KUKA KRL program: EPS_2_251825_SA32_A_20260116064114.src

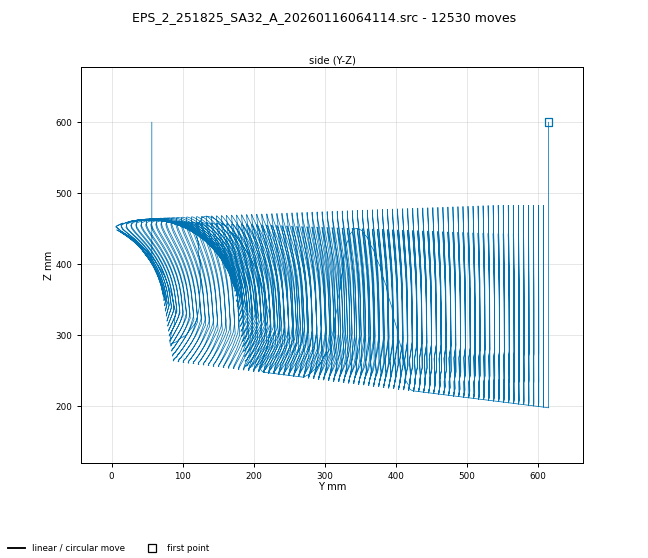
[picture p0: tool path of EPS_2_251825_SA32_A_20260116064114.src, 12530 of 12532 moves have a stored position in this frame; points joined in program order, loops and branches not executed]
&ACCESS RVP
&REL 4
&COMMENT QRS 19112012
&PARAM EDITMASK = *
DEF PART()
EXT BAS (BAS_COMMAND :IN,REAL :IN )
INT I
BAS (#INITMOV,0 )

;KUKA QRS Post kuka4.cps  Date:22-06-2017 !

File_ID=2979

QRS_PRE_INIT()

;Init var - Until changes are made in qrs_pre_init
Outlet_Square_prg=0
Inlet_1_Square_prg=0
Inlet_2_Square_prg=0
Inlet_3_Square_prg=0
Inlet_4_Square_prg=0
Inlet_5_Square_prg=0

Outlet_1={X 0.000, Y 540.910, Z 382.500, B 0.000, E1 0.000 }
Inlet_1={X 0.000, Y 543.760, Z 342.500, B 0.000, E1 213.000 }
Outlet_1_type=201
Inlet_1_type=201
;QRS#1=Sidecore dimensions
;QRS#2=200-8" PVC SDR 35
;QRS#3=200-8" PVC SDR 35
;QRS#4=
;QRS#5=
;QRS#6=
;QRS#7=
;QRS#8=
;QRS#9=12-08 PSX
;QRS#10=12-08 PSX
;QRS#11=
;QRS#12=
;QRS#13=
;QRS#14=
;QRS#15=
;QRS#16=1220x127x762 2,5'
;QRS#17=EPS Height
;QRS#18=483
;QRS#19=*
;QRS#20= UPDATED VERSION 22-06-2017
;QRS#21=*
Outlet_Square=0100
Inlet_1_Square=0100
Inlet_2_Square=0
Inlet_3_Square=0
Inlet_4_Square=0
Inlet_5_Square=0
Mill_Square=1
Outlet_Square_Prg=204
Inlet_1_Square_prg=204

QRS_INIT()

$ADVANCE=5

; T1
PTP {E1 173.659,E2 173.659}
PTP {X 0,Y 615.41,A -85,B 0,C 180,E1 173.659,E2 173.659,E3 0,E4 0,E5 0,E6 0}
QRS_SPEED_INIT()
LIN {X 0,Y 615.41,Z 600,A -85,B 0,C 180,E1 173.659,E2 173.659,E3 0,E4 0,E5 0,E6 0} C_VEL
LIN {X 0,Y 615.41,Z 207.878,A -85,B 0,C 180,E1 173.659,E2 173.659} C_VEL
LIN {X 0,Y 615.41,Z 199.7,A -85,B 0,C 180,E1 173.659,E2 173.659} C_VEL
LIN {X 0,Y 615.409,Z 197.7,A -85,B 0,C 180,E1 173.473,E2 173.473} C_VEL
LIN {X 0,Y 615.46,Z 197.7,A -85,B 0,C 180,E1 170.805,E2 170.805} C_VEL
LIN {X 0,Y 615.441,Z 197.7,A -85,B 0,C 180,E1 168.143,E2 168.143} C_VEL
LIN {X 0,Y 615.434,Z 197.7,A -85,B 0,C 180,E1 166.082,E2 166.082} C_VEL
LIN {X 0,Y 615.409,Z 197.7,A -85,B 0,C 180,E1 163.589,E2 163.589} C_VEL
LIN {X 0,Y 615.415,Z 197.7,A -85,B 0,C 180,E1 161.357,E2 161.357} C_VEL
LIN {X 0,Y 615.492,Z 197.701,A -85,B 0,C 180,E1 158.574,E2 158.574} C_VEL
LIN {X 0,Y 615.407,Z 197.7,A -85,B 0,C 180,E1 155.73,E2 155.73} C_VEL
LIN {X 0,Y 615.41,Z 197.7,A -85,B 0,C 180,E1 153.558,E2 153.558} C_VEL
LIN {X 0,Y 615.479,Z 197.703,A -85,B 0,C 180,E1 150.599,E2 150.599} C_VEL
LIN {X 0,Y 615.449,Z 197.7,A -85,B 0,C 180,E1 148.319,E2 148.319} C_VEL
LIN {X 0,Y 615.418,Z 197.7,A -85,B 0,C 180,E1 145.98,E2 145.98} C_VEL
LIN {X 0,Y 615.411,Z 197.699,A -85,B 0,C 180,E1 143.577,E2 143.577} C_VEL
LIN {X 0,Y 615.465,Z 197.699,A -85,B 0,C 180,E1 140.939,E2 140.939} C_VEL
LIN {X 0,Y 615.472,Z 197.7,A -85,B 0,C 180,E1 138.533,E2 138.533} C_VEL
LIN {X 0,Y 615.417,Z 197.7,A -85,B 0,C 180,E1 136.008,E2 136.008} C_VEL
LIN {X 0,Y 615.416,Z 197.7,A -85,B 0,C 180,E1 133.999,E2 133.999} C_VEL
LIN {X 0,Y 615.418,Z 197.699,A -85,B 0,C 180,E1 131.478,E2 131.478} C_VEL
LIN {X 0,Y 615.473,Z 197.701,A -85,B 0,C 180,E1 128.904,E2 128.904} C_VEL
LIN {X 0,Y 615.449,Z 197.7,A -85,B 0,C 180,E1 126.426,E2 126.426} C_VEL
LIN {X 0,Y 615.413,Z 197.7,A -85,B 0,C 180,E1 124.026,E2 124.026} C_VEL
LIN {X 0,Y 615.412,Z 197.699,A -85,B 0,C 180,E1 121.689,E2 121.689} C_VEL
LIN {X 0,Y 615.427,Z 197.699,A -85,B 0,C 180,E1 119.409,E2 119.409} C_VEL
LIN {X 0,Y 615.445,Z 197.7,A -85,B 0,C 180,E1 116.445,E2 116.445} C_VEL
LIN {X 0,Y 615.413,Z 197.699,A -85,B 0,C 180,E1 114.01,E2 114.01} C_VEL
LIN {X 0,Y 615.418,Z 197.7,A -85,B 0,C 180,E1 112.138,E2 112.138} C_VEL
LIN {X 0,Y 615.412,Z 197.7,A -85,B 0,C 180,E1 110.035,E2 110.035} C_VEL
LIN {X 0,Y 615.41,Z 197.7,A -85,B 0,C 180,E1 107.959,E2 107.959} C_VEL
LIN {X 0,Y 615.453,Z 197.699,A -85,B 0,C 180,E1 105.227,E2 105.227} C_VEL
LIN {X 0,Y 615.442,Z 197.701,A -85,B 0,C 180,E1 102.531,E2 102.531} C_VEL
LIN {X 0,Y 615.445,Z 197.7,A -85,B 0,C 180,E1 100.527,E2 100.527} C_VEL
LIN {X 0,Y 615.41,Z 197.7,A -85,B 0,C 180,E1 97.876,E2 97.876} C_VEL
LIN {X 0,Y 615.458,Z 197.699,A -85,B 0,C 180,E1 95.241,E2 95.241} C_VEL
LIN {X 0,Y 615.451,Z 197.7,A -85,B 0,C 180,E1 92.618,E2 92.618} C_VEL
LIN {X 0,Y 615.412,Z 197.699,A -85,B 0,C 180,E1 90,E2 90} C_VEL
LIN {X 0,Y 615.447,Z 197.699,A -85,B 0,C 180,E1 87.382,E2 87.382} C_VEL
LIN {X 0,Y 615.463,Z 197.7,A -85,B 0,C 180,E1 84.759,E2 84.759} C_VEL
LIN {X 0,Y 615.413,Z 197.699,A -85,B 0,C 180,E1 82.124,E2 82.124} C_VEL
LIN {X 0,Y 615.413,Z 197.699,A -85,B 0,C 180,E1 80.137,E2 80.137} C_VEL
LIN {X 0,Y 615.413,Z 197.699,A -85,B 0,C 180,E1 78.138,E2 78.138} C_VEL
LIN {X 0,Y 615.431,Z 197.809,A -85,B 0,C 180,E1 75.604,E2 75.604} C_VEL
LIN {X 0,Y 615.454,Z 214.764,A -85,B 0,C 180,E1 72.729,E2 72.729} C_VEL
LIN {X 0,Y 615.44,Z 229.187,A -85,B 0,C 180,E1 70.314,E2 70.314} C_VEL
LIN {X 0,Y 615.464,Z 232.183,A -85,B 0,C 180,E1 69.813,E2 69.813} C_VEL
LIN {X 0,Y 615.455,Z 338.803,A -85,B 0,C 180,E1 68.546,E2 68.546} C_VEL
LIN {X 0,Y 615.454,Z 351.86,A -85,B 0,C 180,E1 68.26,E2 68.26} C_VEL
LIN {X 0,Y 615.477,Z 364.037,A -85,B 0,C 180,E1 67.864,E2 67.864} C_VEL
LIN {X 0,Y 615.493,Z 376.068,A -85,B 0,C 180,E1 67.336,E2 67.336} C_VEL
LIN {X 0,Y 615.484,Z 387.07,A -85,B 0,C 180,E1 66.712,E2 66.712} C_VEL
LIN {X 0,Y 615.499,Z 397.482,A -85,B 0,C 180,E1 65.973,E2 65.973} C_VEL
LIN {X 0,Y 615.498,Z 406.502,A -85,B 0,C 180,E1 65.19,E2 65.19} C_VEL
LIN {X 0,Y 615.494,Z 415.026,A -85,B 0,C 180,E1 64.285,E2 64.285} C_VEL
LIN {X 0,Y 615.498,Z 422.868,A -85,B 0,C 180,E1 63.249,E2 63.249} C_VEL
LIN {X 0,Y 615.498,Z 428.792,A -85,B 0,C 180,E1 62.271,E2 62.271} C_VEL
LIN {X 0,Y 615.496,Z 433.284,A -85,B 0,C 180,E1 61.343,E2 61.343} C_VEL
LIN {X 0,Y 615.497,Z 437.518,A -85,B 0,C 180,E1 60.19,E2 60.19} C_VEL
LIN {X 0,Y 615.495,Z 440.638,A -85,B 0,C 180,E1 58.9,E2 58.9} C_VEL
LIN {X 0,Y 615.496,Z 442.14,A -85,B 0,C 180,E1 57.656,E2 57.656} C_VEL
LIN {X 0,Y 615.493,Z 442.273,A -85,B 0,C 180,E1 56.453,E2 56.453} C_VEL
LIN {X 0,Y 615.5,Z 440.932,A -85,B 0,C 180,E1 55.187,E2 55.187} C_VEL
LIN {X 0,Y 615.496,Z 438.744,A -85,B 0,C 180,E1 54.154,E2 54.154} C_VEL
LIN {X 0,Y 615.492,Z 435.237,A -85,B 0,C 180,E1 53.052,E2 53.052} C_VEL
LIN {X 0,Y 615.494,Z 430.341,A -85,B 0,C 180,E1 51.933,E2 51.933} C_VEL
LIN {X 0,Y 615.496,Z 424.633,A -85,B 0,C 180,E1 50.927,E2 50.927} C_VEL
LIN {X 0,Y 615.497,Z 417.282,A -85,B 0,C 180,E1 49.9,E2 49.9} C_VEL
LIN {X 0,Y 615.493,Z 408.29,A -85,B 0,C 180,E1 48.895,E2 48.895} C_VEL
LIN {X 0,Y 615.499,Z 399.11,A -85,B 0,C 180,E1 48.065,E2 48.065} C_VEL
LIN {X 0,Y 615.494,Z 388.597,A -85,B 0,C 180,E1 47.298,E2 47.298} C_VEL
LIN {X 0,Y 615.477,Z 377.738,A -85,B 0,C 180,E1 46.661,E2 46.661} C_VEL
LIN {X 0,Y 615.491,Z 366.43,A -85,B 0,C 180,E1 46.139,E2 46.139} C_VEL
LIN {X 0,Y 615.477,Z 353.773,A -85,B 0,C 180,E1 45.703,E2 45.703} C_VEL
LIN {X 0,Y 615.488,Z 341.141,A -85,B 0,C 180,E1 45.408,E2 45.408} C_VEL
LIN {X 0,Y 615.485,Z 319.264,A -85,B 0,C 180,E1 45.122,E2 45.122} C_VEL
LIN {X 0,Y 615.477,Z 232.126,A -85,B 0,C 180,E1 44.088,E2 44.088} C_VEL
LIN {X 0,Y 615.495,Z 215.346,A -85,B 0,C 180,E1 41.281,E2 41.281} C_VEL
LIN {X 0,Y 615.457,Z 198.823,A -85,B 0,C 180,E1 38.48,E2 38.48} C_VEL
LIN {X 0,Y 615.445,Z 197.695,A -85,B 0,C 180,E1 38.272,E2 38.272} C_VEL
LIN {X 0,Y 615.464,Z 197.689,A -85,B 0,C 180,E1 35.61,E2 35.61} C_VEL
LIN {X 0,Y 615.495,Z 197.691,A -85,B 0,C 180,E1 33.229,E2 33.229} C_VEL
LIN {X 0,Y 615.487,Z 197.702,A -85,B 0,C 180,E1 30.913,E2 30.913} C_VEL
LIN {X 0,Y 615.447,Z 197.696,A -85,B 0,C 180,E1 28.446,E2 28.446} C_VEL
LIN {X 0,Y 615.446,Z 197.696,A -85,B 0,C 180,E1 26.44,E2 26.44} C_VEL
LIN {X 0,Y 615.441,Z 197.693,A -85,B 0,C 180,E1 24.002,E2 24.002} C_VEL
LIN {X 0,Y 615.492,Z 197.689,A -85,B 0,C 180,E1 21.426,E2 21.426} C_VEL
LIN {X 0,Y 615.449,Z 197.697,A -85,B 0,C 180,E1 18.599,E2 18.599} C_VEL
LIN {X 0,Y 615.438,Z 197.696,A -85,B 0,C 180,E1 16.421,E2 16.421} C_VEL
LIN {X 0,Y 615.443,Z 197.696,A -85,B 0,C 180,E1 14.545,E2 14.545} C_VEL
LIN {X 0,Y 615.441,Z 197.696,A -85,B 0,C 180,E1 12.527,E2 12.527} C_VEL
LIN {X 0,Y 615.439,Z 197.696,A -85,B 0,C 180,E1 10.523,E2 10.523} C_VEL
LIN {X 0,Y 615.439,Z 197.696,A -85,B 0,C 180,E1 8.533,E2 8.533} C_VEL
LIN {X 0,Y 615.438,Z 197.696,A -85,B 0,C 180,E1 6.552,E2 6.552} C_VEL
LIN {X 0,Y 615.437,Z 197.697,A -85,B 0,C 180,E1 4.581,E2 4.581} C_VEL
LIN {X 0,Y 615.439,Z 197.697,A -85,B 0,C 180,E1 2.614,E2 2.614} C_VEL
LIN {X 0,Y 615.439,Z 197.697,A -85,B 0,C 180,E1 0.651,E2 0.651} C_VEL
LIN {X 0,Y 615.439,Z 197.697,A -85,B 0,C 180,E1 -1.312,E2 -1.312} C_VEL
LIN {X 0,Y 615.441,Z 197.697,A -85,B 0,C 180,E1 -3.277,E2 -3.277} C_VEL
LIN {X 0,Y 615.441,Z 197.697,A -85,B 0,C 180,E1 -5.245,E2 -5.245} C_VEL
LIN {X 0,Y 615.441,Z 197.697,A -85,B 0,C 180,E1 -7.22,E2 -7.22} C_VEL
LIN {X 0,Y 615.44,Z 197.698,A -85,B 0,C 180,E1 -9.203,E2 -9.203} C_VEL
LIN {X 0,Y 615.439,Z 197.698,A -85,B 0,C 180,E1 -11.197,E2 -11.197} C_VEL
LIN {X 0,Y 615.436,Z 197.698,A -85,B 0,C 180,E1 -13.205,E2 -13.205} C_VEL
LIN {X 0,Y 615.434,Z 197.697,A -85,B 0,C 180,E1 -15.23,E2 -15.23} C_VEL
LIN {X 0,Y 615.431,Z 197.697,A -85,B 0,C 180,E1 -17.275,E2 -17.275} C_VEL
LIN {X 0,Y 615.427,Z 197.697,A -85,B 0,C 180,E1 -19.343,E2 -19.343} C_VEL
LIN {X 0,Y 615.425,Z 197.697,A -85,B 0,C 180,E1 -21.437,E2 -21.437} C_VEL
LIN {X 0,Y 615.447,Z 197.696,A -85,B 0,C 180,E1 -24.003,E2 -24.003} C_VEL
LIN {X 0,Y 615.493,Z 197.699,A -85,B 0,C 180,E1 -26.446,E2 -26.446} C_VEL
LIN {X 0,Y 615.471,Z 197.701,A -85,B 0,C 180,E1 -28.661,E2 -28.661} C_VEL
LIN {X 0,Y 615.431,Z 197.698,A -85,B 0,C 180,E1 -31.08,E2 -31.08} C_VEL
LIN {X 0,Y 615.423,Z 197.698,A -85,B 0,C 180,E1 -33.242,E2 -33.242} C_VEL
LIN {X 0,Y 615.439,Z 197.696,A -85,B 0,C 180,E1 -35.83,E2 -35.83} C_VEL
LIN {X 0,Y 615.468,Z 197.696,A -85,B 0,C 180,E1 -38.072,E2 -38.072} C_VEL
LIN {X 0,Y 615.467,Z 197.7,A -85,B 0,C 180,E1 -40.61,E2 -40.61} C_VEL
LIN {X 0,Y 615.421,Z 197.699,A -85,B 0,C 180,E1 -43.042,E2 -43.042} C_VEL
LIN {X 0,Y 615.422,Z 197.699,A -85,B 0,C 180,E1 -45.076,E2 -45.076} C_VEL
LIN {X 0,Y 615.455,Z 197.697,A -85,B 0,C 180,E1 -47.925,E2 -47.925} C_VEL
LIN {X 0,Y 615.496,Z 197.699,A -85,B 0,C 180,E1 -50.252,E2 -50.252} C_VEL
LIN {X 0,Y 615.417,Z 197.699,A -85,B 0,C 180,E1 -53.074,E2 -53.074} C_VEL
LIN {X 0,Y 615.415,Z 197.699,A -85,B 0,C 180,E1 -55.311,E2 -55.311} C_VEL
LIN {X 0,Y 615.434,Z 197.699,A -85,B 0,C 180,E1 -57.679,E2 -57.679} C_VEL
LIN {X 0,Y 615.442,Z 197.7,A -85,B 0,C 180,E1 -60.592,E2 -60.592} C_VEL
LIN {X 0,Y 615.415,Z 197.7,A -85,B 0,C 180,E1 -62.97,E2 -62.97} C_VEL
LIN {X 0,Y 615.413,Z 197.7,A -85,B 0,C 180,E1 -65.006,E2 -65.006} C_VEL
LIN {X 0,Y 615.419,Z 197.809,A -85,B 0,C 180,E1 -67.442,E2 -67.442} C_VEL
LIN {X 0,Y 615.495,Z 217.695,A -85,B 0,C 180,E1 -70.142,E2 -70.142} C_VEL
LIN {X 0,Y 615.456,Z 238.373,A -85,B 0,C 180,E1 -72.9,E2 -72.9} C_VEL
LIN {X 0,Y 615.478,Z 258.907,A -85,B 0,C 180,E1 -75.605,E2 -75.605} C_VEL
LIN {X 0,Y 615.454,Z 270.473,A -85,B 0,C 180,E1 -77.113,E2 -77.113} C_VEL
LIN {X 0,Y 615.473,Z 378.853,A -85,B 0,C 180,E1 -78.411,E2 -78.411} C_VEL
LIN {X 0,Y 615.467,Z 391.36,A -85,B 0,C 180,E1 -78.682,E2 -78.682} C_VEL
LIN {X 0,Y 615.485,Z 404.67,A -85,B 0,C 180,E1 -79.115,E2 -79.115} C_VEL
LIN {X 0,Y 615.484,Z 416.484,A -85,B 0,C 180,E1 -79.64,E2 -79.64} C_VEL
LIN {X 0,Y 615.493,Z 427.999,A -85,B 0,C 180,E1 -80.304,E2 -80.304} C_VEL
LIN {X 0,Y 615.499,Z 438.345,A -85,B 0,C 180,E1 -81.05,E2 -81.05} C_VEL
LIN {X 0,Y 615.497,Z 446.814,A -85,B 0,C 180,E1 -81.794,E2 -81.794} C_VEL
LIN {X 0,Y 615.498,Z 454.608,A -85,B 0,C 180,E1 -82.62,E2 -82.62} C_VEL
LIN {X 0,Y 615.496,Z 462.204,A -85,B 0,C 180,E1 -83.608,E2 -83.608} C_VEL
LIN {X 0,Y 615.498,Z 469.205,A -85,B 0,C 180,E1 -84.759,E2 -84.759} C_VEL
LIN {X 0,Y 615.494,Z 473.852,A -85,B 0,C 180,E1 -85.744,E2 -85.744} C_VEL
LIN {X 0,Y 615.494,Z 477.399,A -85,B 0,C 180,E1 -86.727,E2 -86.727} C_VEL
LIN {X 0,Y 615.497,Z 479.233,A -85,B 0,C 180,E1 -87.382,E2 -87.382} C_VEL
LIN {X 0,Y 615.499,Z 480.608,A -85,B 0,C 180,E1 -88.037,E2 -88.037} C_VEL
LIN {X 0,Y 615.496,Z 482.174,A -85,B 0,C 180,E1 -89.346,E2 -89.346} C_VEL
LIN {X 0,Y 615.494,Z 482.389,A -85,B 0,C 180,E1 -90,E2 -90} C_VEL
LIN {X 0,Y 615.495,Z 481.58,A -85,B 0,C 180,E1 -91.309,E2 -91.309} C_VEL
LIN {X 0,Y 615.499,Z 480.608,A -85,B 0,C 180,E1 -91.963,E2 -91.963} C_VEL
LIN {X 0,Y 615.497,Z 479.233,A -85,B 0,C 180,E1 -92.618,E2 -92.618} C_VEL
LIN {X 0,Y 615.496,Z 476.35,A -85,B 0,C 180,E1 -93.601,E2 -93.601} C_VEL
LIN {X 0,Y 615.498,Z 472.442,A -85,B 0,C 180,E1 -94.584,E2 -94.584} C_VEL
LIN {X 0,Y 615.499,Z 467.405,A -85,B 0,C 180,E1 -95.57,E2 -95.57} C_VEL
LIN {X 0,Y 615.497,Z 460.875,A -85,B 0,C 180,E1 -96.583,E2 -96.583} C_VEL
LIN {X 0,Y 615.497,Z 453.134,A -85,B 0,C 180,E1 -97.545,E2 -97.545} C_VEL
LIN {X 0,Y 615.498,Z 445.047,A -85,B 0,C 180,E1 -98.371,E2 -98.371} C_VEL
LIN {X 0,Y 615.499,Z 435.17,A -85,B 0,C 180,E1 -99.198,E2 -99.198} C_VEL
LIN {X 0,Y 615.492,Z 423.984,A -85,B 0,C 180,E1 -99.945,E2 -99.945} C_VEL
LIN {X 0,Y 615.486,Z 413.028,A -85,B 0,C 180,E1 -100.527,E2 -100.527} C_VEL
LIN {X 0,Y 615.475,Z 400.523,A -85,B 0,C 180,E1 -101.039,E2 -101.039} C_VEL
LIN {X 0,Y 615.467,Z 388.081,A -85,B 0,C 180,E1 -101.402,E2 -101.402} C_VEL
LIN {X 0,Y 615.472,Z 374.489,A -85,B 0,C 180,E1 -101.652,E2 -101.652} C_VEL
LIN {X 0,Y 615.454,Z 270.473,A -85,B 0,C 180,E1 -102.887,E2 -102.887} C_VEL
LIN {X 0,Y 615.479,Z 249.991,A -85,B 0,C 180,E1 -105.565,E2 -105.565} C_VEL
LIN {X 0,Y 615.468,Z 228.307,A -85,B 0,C 180,E1 -108.438,E2 -108.438} C_VEL
LIN {X 0,Y 615.461,Z 209.935,A -85,B 0,C 180,E1 -110.906,E2 -110.906} C_VEL
LIN {X 0,Y 615.416,Z 197.7,A -85,B 0,C 180,E1 -112.59,E2 -112.59} C_VEL
LIN {X 0,Y 615.411,Z 197.7,A -85,B 0,C 180,E1 -114.994,E2 -114.994} C_VEL
LIN {X 0,Y 615.42,Z 197.7,A -85,B 0,C 180,E1 -117.18,E2 -117.18} C_VEL
LIN {X 0,Y 615.45,Z 197.7,A -85,B 0,C 180,E1 -120.161,E2 -120.161} C_VEL
LIN {X 0,Y 615.421,Z 197.7,A -85,B 0,C 180,E1 -122.461,E2 -122.461} C_VEL
LIN {X 0,Y 615.409,Z 197.7,A -85,B 0,C 180,E1 -124.819,E2 -124.819} C_VEL
LIN {X 0,Y 615.426,Z 197.7,A -85,B 0,C 180,E1 -127.245,E2 -127.245} C_VEL
LIN {X 0,Y 615.453,Z 197.7,A -85,B 0,C 180,E1 -130.083,E2 -130.083} C_VEL
LIN {X 0,Y 615.423,Z 197.7,A -85,B 0,C 180,E1 -132.357,E2 -132.357} C_VEL
LIN {X 0,Y 615.411,Z 197.7,A -85,B 0,C 180,E1 -134.923,E2 -134.923} C_VEL
LIN {X 0,Y 615.413,Z 197.7,A -85,B 0,C 180,E1 -136.958,E2 -136.958} C_VEL
LIN {X 0,Y 615.449,Z 197.7,A -85,B 0,C 180,E1 -139.389,E2 -139.389} C_VEL
LIN {X 0,Y 615.456,Z 197.7,A -85,B 0,C 180,E1 -141.99,E2 -141.99} C_VEL
LIN {X 0,Y 615.418,Z 197.7,A -85,B 0,C 180,E1 -144.377,E2 -144.377} C_VEL
LIN {X 0,Y 615.409,Z 197.7,A -85,B 0,C 180,E1 -146.757,E2 -146.757} C_VEL
LIN {X 0,Y 615.423,Z 197.7,A -85,B 0,C 180,E1 -149.074,E2 -149.074} C_VEL
LIN {X 0,Y 615.482,Z 197.7,A -85,B 0,C 180,E1 -151.548,E2 -151.548} C_VEL
LIN {X 0,Y 615.421,Z 197.7,A -85,B 0,C 180,E1 -154.279,E2 -154.279} C_VEL
LIN {X 0,Y 615.412,Z 197.7,A -85,B 0,C 180,E1 -156.438,E2 -156.438} C_VEL
LIN {X 0,Y 615.409,Z 197.7,A -85,B 0,C 180,E1 -158.563,E2 -158.563} C_VEL
LIN {X 0,Y 615.409,Z 197.7,A -85,B 0,C 180,E1 -160.657,E2 -160.657} C_VEL
LIN {X 0,Y 615.48,Z 197.703,A -85,B 0,C 180,E1 -163.566,E2 -163.566} C_VEL
LIN {X 0,Y 615.428,Z 197.7,A -85,B 0,C 180,E1 -166.122,E2 -166.122} C_VEL
LIN {X 0,Y 615.426,Z 197.7,A -85,B 0,C 180,E1 -168.135,E2 -168.135} C_VEL
LIN {X 0,Y 615.425,Z 197.7,A -85,B 0,C 180,E1 -170.134,E2 -170.134} C_VEL
LIN {X 0,Y 615.426,Z 197.7,A -85,B 0,C 180,E1 -172.12,E2 -172.12} C_VEL
LIN {X 0,Y 615.427,Z 197.7,A -85,B 0,C 180,E1 -174.098,E2 -174.098} C_VEL
LIN {X 0,Y 615.428,Z 197.7,A -85,B 0,C 180,E1 -176.068,E2 -176.068} C_VEL
LIN {X 0,Y 615.431,Z 197.7,A -85,B 0,C 180,E1 -178.033,E2 -178.033} C_VEL
LIN {X 0,Y 615.433,Z 197.7,A -85,B 0,C 180,E1 -179.996,E2 -179.996} C_VEL
LIN {X 0,Y 615.436,Z 197.7,A -85,B 0,C 180,E1 -181.959,E2 -181.959} C_VEL
LIN {X 0,Y 615.438,Z 197.7,A -85,B 0,C 180,E1 -183.925,E2 -183.925} C_VEL
LIN {X 0,Y 615.409,Z 197.7,A -85,B 0,C 180,E1 -186.527,E2 -186.527} C_VEL
LIN {X 0,Y 614.766,Z 197.848,A -85,B 0,C 180,E1 -187.073,E2 -187.073} C_VEL
LIN {X 0,Y 611.963,Z 198.253,A -85,B 0,C 180,E1 -187.959,E2 -187.959} C_VEL
LIN {X 0,Y 609.573,Z 198.567,A -85,B 0,C 180,E1 -188.672,E2 -188.672} C_VEL
LIN {X 0,Y 608.526,Z 198.688,A -85,B 0,C 180,E1 -189.222,E2 -189.222} C_VEL
LIN {X 0,Y 608.43,Z 198.696,A -85,B 0,C 180,E1 -189.408,E2 -189.408} C_VEL
LIN {X 0,Y 608.413,Z 198.694,A -85,B 0,C 180,E1 -191.996,E2 -191.996} C_VEL
LIN {X 0,Y 608.395,Z 198.696,A -85,B 0,C 180,E1 -194.034,E2 -194.034} C_VEL
LIN {X 0,Y 608.381,Z 198.696,A -85,B 0,C 180,E1 -196.506,E2 -196.506} C_VEL
LIN {X 0,Y 608.413,Z 198.694,A -85,B 0,C 180,E1 -198.866,E2 -198.866} C_VEL
LIN {X 0,Y 608.444,Z 198.694,A -85,B 0,C 180,E1 -201.687,E2 -201.687} C_VEL
LIN {X 0,Y 608.394,Z 198.695,A -85,B 0,C 180,E1 -204.568,E2 -204.568} C_VEL
LIN {X 0,Y 608.451,Z 198.695,A -85,B 0,C 180,E1 -207.205,E2 -207.205} C_VEL
LIN {X 0,Y 608.396,Z 198.696,A -85,B 0,C 180,E1 -209.962,E2 -209.962} C_VEL
LIN {X 0,Y 608.391,Z 198.695,A -85,B 0,C 180,E1 -212.514,E2 -212.514} C_VEL
LIN {X 0,Y 608.4,Z 198.697,A -85,B 0,C 180,E1 -214.901,E2 -214.901} C_VEL
LIN {X 0,Y 608.421,Z 198.695,A -85,B 0,C 180,E1 -217.742,E2 -217.742} C_VEL
LIN {X 0,Y 608.382,Z 198.696,A -85,B 0,C 180,E1 -220.323,E2 -220.323} C_VEL
LIN {X 0,Y 608.424,Z 198.696,A -85,B 0,C 180,E1 -222.954,E2 -222.954} C_VEL
LIN {X 0,Y 608.4,Z 198.697,A -85,B 0,C 180,E1 -225.733,E2 -225.733} C_VEL
LIN {X 0,Y 608.401,Z 198.695,A -85,B 0,C 180,E1 -227.935,E2 -227.935} C_VEL
LIN {X 0,Y 608.428,Z 198.693,A -85,B 0,C 180,E1 -230.697,E2 -230.697} C_VEL
LIN {X 0,Y 608.434,Z 198.698,A -85,B 0,C 180,E1 -233.085,E2 -233.085} C_VEL
LIN {X 0,Y 608.441,Z 198.694,A -85,B 0,C 180,E1 -235.53,E2 -235.53} C_VEL
LIN {X 0,Y 608.409,Z 198.694,A -85,B 0,C 180,E1 -237.903,E2 -237.903} C_VEL
LIN {X 0,Y 608.396,Z 198.694,A -85,B 0,C 180,E1 -240.217,E2 -240.217} C_VEL
LIN {X 0,Y 608.44,Z 198.693,A -85,B 0,C 180,E1 -242.785,E2 -242.785} C_VEL
LIN {X 0,Y 608.411,Z 198.693,A -85,B 0,C 180,E1 -245.845,E2 -245.845} C_VEL
LIN {X 0,Y 608.406,Z 198.693,A -85,B 0,C 180,E1 -248.307,E2 -248.307} C_VEL
LIN {X 0,Y 608.431,Z 198.701,A -85,B 0,C 180,E1 -251.13,E2 -251.13} C_VEL
LIN {X 0,Y 608.396,Z 198.695,A -85,B 0,C 180,E1 -253.905,E2 -253.905} C_VEL
LIN {X 0,Y 608.42,Z 198.694,A -85,B 0,C 180,E1 -256.643,E2 -256.643} C_VEL
LIN {X 0,Y 608.431,Z 198.696,A -85,B 0,C 180,E1 -259.35,E2 -259.35} C_VEL
LIN {X 0,Y 608.406,Z 198.693,A -85,B 0,C 180,E1 -262.032,E2 -262.032} C_VEL
LIN {X 0,Y 608.431,Z 198.694,A -85,B 0,C 180,E1 -264.698,E2 -264.698} C_VEL
LIN {X 0,Y 608.439,Z 198.694,A -85,B 0,C 180,E1 -267.352,E2 -267.352} C_VEL
LIN {X 0,Y 608.403,Z 198.693,A -85,B 0,C 180,E1 -270,E2 -270} C_VEL
LIN {X 0,Y 608.436,Z 198.694,A -85,B 0,C 180,E1 -272.648,E2 -272.648} C_VEL
LIN {X 0,Y 608.435,Z 198.695,A -85,B 0,C 180,E1 -275.302,E2 -275.302} C_VEL
LIN {X 0,Y 608.408,Z 198.693,A -85,B 0,C 180,E1 -277.968,E2 -277.968} C_VEL
LIN {X 0,Y 608.429,Z 198.695,A -85,B 0,C 180,E1 -280.65,E2 -280.65} C_VEL
LIN {X 0,Y 608.426,Z 198.695,A -85,B 0,C 180,E1 -283.357,E2 -283.357} C_VEL
LIN {X 0,Y 608.438,Z 198.817,A -85,B 0,C 180,E1 -284.336,E2 -284.336} C_VEL
LIN {X 0,Y 608.443,Z 216.169,A -85,B 0,C 180,E1 -287.303,E2 -287.303} C_VEL
LIN {X 0,Y 608.419,Z 230.661,A -85,B 0,C 180,E1 -289.747,E2 -289.747} C_VEL
LIN {X 0,Y 608.43,Z 232.362,A -85,B 0,C 180,E1 -290.032,E2 -290.032} C_VEL
LIN {X 0,Y 608.536,Z 331.818,A -85,B 0,C 180,E1 -291.222,E2 -291.222} C_VEL
LIN {X 0,Y 608.503,Z 345.333,A -85,B 0,C 180,E1 -291.445,E2 -291.445} C_VEL
LIN {X 0,Y 608.492,Z 359.013,A -85,B 0,C 180,E1 -291.824,E2 -291.824} C_VEL
LIN {X 0,Y 608.506,Z 371.463,A -85,B 0,C 180,E1 -292.314,E2 -292.314} C_VEL
LIN {X 0,Y 608.483,Z 383.511,A -85,B 0,C 180,E1 -292.945,E2 -292.945} C_VEL
LIN {X 0,Y 608.497,Z 394.341,A -85,B 0,C 180,E1 -293.662,E2 -293.662} C_VEL
LIN {X 0,Y 608.478,Z 403.986,A -85,B 0,C 180,E1 -294.45,E2 -294.45} C_VEL
LIN {X 0,Y 608.451,Z 412.483,A -85,B 0,C 180,E1 -295.3,E2 -295.3} C_VEL
LIN {X 0,Y 608.46,Z 420.032,A -85,B 0,C 180,E1 -296.218,E2 -296.218} C_VEL
LIN {X 0,Y 608.453,Z 426.713,A -85,B 0,C 180,E1 -297.217,E2 -297.217} C_VEL
LIN {X 0,Y 608.441,Z 432.294,A -85,B 0,C 180,E1 -298.266,E2 -298.266} C_VEL
LIN {X 0,Y 608.426,Z 436.889,A -85,B 0,C 180,E1 -299.4,E2 -299.4} C_VEL
LIN {X 0,Y 608.446,Z 440.145,A -85,B 0,C 180,E1 -300.545,E2 -300.545} C_VEL
LIN {X 0,Y 608.441,Z 441.63,A -85,B 0,C 180,E1 -301.317,E2 -301.317} C_VEL
LIN {X 0,Y 608.421,Z 442.879,A -85,B 0,C 180,E1 -302.529,E2 -302.529} C_VEL
LIN {X 0,Y 608.416,Z 442.761,A -85,B 0,C 180,E1 -303.739,E2 -303.739} C_VEL
LIN {X 0,Y 608.424,Z 441.396,A -85,B 0,C 180,E1 -304.913,E2 -304.913} C_VEL
LIN {X 0,Y 608.443,Z 438.748,A -85,B 0,C 180,E1 -306.091,E2 -306.091} C_VEL
LIN {X 0,Y 608.43,Z 435.136,A -85,B 0,C 180,E1 -307.164,E2 -307.164} C_VEL
LIN {X 0,Y 608.431,Z 430.227,A -85,B 0,C 180,E1 -308.246,E2 -308.246} C_VEL
LIN {X 0,Y 608.441,Z 424.013,A -85,B 0,C 180,E1 -309.304,E2 -309.304} C_VEL
LIN {X 0,Y 608.457,Z 416.373,A -85,B 0,C 180,E1 -310.339,E2 -310.339} C_VEL
LIN {X 0,Y 608.452,Z 408.826,A -85,B 0,C 180,E1 -311.175,E2 -311.175} C_VEL
LIN {X 0,Y 608.495,Z 399.125,A -85,B 0,C 180,E1 -312.057,E2 -312.057} C_VEL
LIN {X 0,Y 608.505,Z 387.951,A -85,B 0,C 180,E1 -312.87,E2 -312.87} C_VEL
LIN {X 0,Y 608.498,Z 376.576,A -85,B 0,C 180,E1 -313.529,E2 -313.529} C_VEL
LIN {X 0,Y 608.507,Z 364.752,A -85,B 0,C 180,E1 -314.058,E2 -314.058} C_VEL
LIN {X 0,Y 608.539,Z 351.382,A -85,B 0,C 180,E1 -314.496,E2 -314.496} C_VEL
LIN {X 0,Y 608.547,Z 338.609,A -85,B 0,C 180,E1 -314.774,E2 -314.774} C_VEL
LIN {X 0,Y 608.463,Z 232.347,A -85,B 0,C 180,E1 -316.059,E2 -316.059} C_VEL
LIN {X 0,Y 608.475,Z 215.893,A -85,B 0,C 180,E1 -318.833,E2 -318.833} C_VEL
LIN {X 0,Y 608.479,Z 200.746,A -85,B 0,C 180,E1 -321.42,E2 -321.42} C_VEL
LIN {X 0,Y 608.416,Z 198.694,A -85,B 0,C 180,E1 -321.794,E2 -321.794} C_VEL
LIN {X 0,Y 608.435,Z 198.69,A -85,B 0,C 180,E1 -323.954,E2 -323.954} C_VEL
LIN {X 0,Y 608.439,Z 198.69,A -85,B 0,C 180,E1 -326.335,E2 -326.335} C_VEL
LIN {X 0,Y 608.451,Z 198.693,A -85,B 0,C 180,E1 -328.729,E2 -328.729} C_VEL
LIN {X 0,Y 608.442,Z 198.693,A -85,B 0,C 180,E1 -331.383,E2 -331.383} C_VEL
LIN {X 0,Y 608.436,Z 198.696,A -85,B 0,C 180,E1 -333.231,E2 -333.231} C_VEL
LIN {X 0,Y 608.435,Z 198.69,A -85,B 0,C 180,E1 -335.853,E2 -335.853} C_VEL
LIN {X 0,Y 608.452,Z 198.689,A -85,B 0,C 180,E1 -338.313,E2 -338.313} C_VEL
LIN {X 0,Y 608.438,Z 198.694,A -85,B 0,C 180,E1 -341.289,E2 -341.289} C_VEL
LIN {X 0,Y 608.418,Z 198.692,A -85,B 0,C 180,E1 -343.91,E2 -343.91} C_VEL
LIN {X 0,Y 608.46,Z 198.693,A -85,B 0,C 180,E1 -346.648,E2 -346.648} C_VEL
LIN {X 0,Y 608.428,Z 198.693,A -85,B 0,C 180,E1 -349.354,E2 -349.354} C_VEL
LIN {X 0,Y 608.443,Z 198.689,A -85,B 0,C 180,E1 -352.037,E2 -352.037} C_VEL
LIN {X 0,Y 608.467,Z 198.694,A -85,B 0,C 180,E1 -354.702,E2 -354.702} C_VEL
LIN {X 0,Y 608.435,Z 198.691,A -85,B 0,C 180,E1 -357.356,E2 -357.356} C_VEL
LIN {X 0,Y 608.437,Z 198.691,A -85,B 0,C 180,E1 -359.342,E2 -359.342} C_VEL
LIN {X 0,Y 608.426,Z 198.692,A -85,B 0,C 180,E1 -361.327,E2 -361.327} C_VEL
LIN {X 0,Y 608.409,Z 198.695,A -85,B 0,C 180,E1 -363.315,E2 -363.315} C_VEL
LIN {X 0,Y 608.422,Z 198.693,A -85,B 0,C 180,E1 -365.306,E2 -365.306} C_VEL
LIN {X 0,Y 608.412,Z 198.694,A -85,B 0,C 180,E1 -367.303,E2 -367.303} C_VEL
LIN {X 0,Y 608.426,Z 198.692,A -85,B 0,C 180,E1 -369.31,E2 -369.31} C_VEL
LIN {X 0,Y 608.411,Z 198.694,A -85,B 0,C 180,E1 -371.328,E2 -371.328} C_VEL
LIN {X 0,Y 608.417,Z 198.692,A -85,B 0,C 180,E1 -373.361,E2 -373.361} C_VEL
LIN {X 0,Y 608.425,Z 198.691,A -85,B 0,C 180,E1 -375.41,E2 -375.41} C_VEL
LIN {X 0,Y 608.407,Z 198.693,A -85,B 0,C 180,E1 -377.481,E2 -377.481} C_VEL
LIN {X 0,Y 608.407,Z 198.693,A -85,B 0,C 180,E1 -379.575,E2 -379.575} C_VEL
LIN {X 0,Y 608.425,Z 198.691,A -85,B 0,C 180,E1 -381.696,E2 -381.696} C_VEL
LIN {X 0,Y 608.434,Z 198.7,A -85,B 0,C 180,E1 -384.574,E2 -384.574} C_VEL
LIN {X 0,Y 608.413,Z 198.693,A -85,B 0,C 180,E1 -387.198,E2 -387.198} C_VEL
LIN {X 0,Y 608.405,Z 198.696,A -85,B 0,C 180,E1 -389.026,E2 -389.026} C_VEL
LIN {X 0,Y 608.404,Z 198.693,A -85,B 0,C 180,E1 -391.322,E2 -391.322} C_VEL
LIN {X 0,Y 608.423,Z 198.692,A -85,B 0,C 180,E1 -393.73,E2 -393.73} C_VEL
LIN {X 0,Y 608.436,Z 198.694,A -85,B 0,C 180,E1 -396.095,E2 -396.095} C_VEL
LIN {X 0,Y 608.405,Z 198.701,A -85,B 0,C 180,E1 -398.595,E2 -398.595} C_VEL
LIN {X 0,Y 608.392,Z 198.695,A -85,B 0,C 180,E1 -401.184,E2 -401.184} C_VEL
LIN {X 0,Y 608.413,Z 198.692,A -85,B 0,C 180,E1 -403.305,E2 -403.305} C_VEL
LIN {X 0,Y 608.449,Z 198.695,A -85,B 0,C 180,E1 -406.13,E2 -406.13} C_VEL
LIN {X 0,Y 608.406,Z 198.696,A -85,B 0,C 180,E1 -408.821,E2 -408.821} C_VEL
LIN {X 0,Y 608.39,Z 198.695,A -85,B 0,C 180,E1 -411.407,E2 -411.407} C_VEL
LIN {X 0,Y 608.44,Z 198.694,A -85,B 0,C 180,E1 -413.957,E2 -413.957} C_VEL
LIN {X 0,Y 608.445,Z 198.698,A -85,B 0,C 180,E1 -416.329,E2 -416.329} C_VEL
LIN {X 0,Y 608.426,Z 198.693,A -85,B 0,C 180,E1 -418.737,E2 -418.737} C_VEL
LIN {X 0,Y 608.388,Z 198.696,A -85,B 0,C 180,E1 -420.977,E2 -420.977} C_VEL
LIN {X 0,Y 608.383,Z 198.696,A -85,B 0,C 180,E1 -423.223,E2 -423.223} C_VEL
LIN {X 0,Y 608.406,Z 198.694,A -85,B 0,C 180,E1 -425.428,E2 -425.428} C_VEL
LIN {X 0,Y 608.415,Z 198.825,A -85,B 0,C 180,E1 -427.309,E2 -427.309} C_VEL
LIN {X 0,Y 608.538,Z 212.666,A -85,B 0,C 180,E1 -429.218,E2 -429.218} C_VEL
LIN {X 0,Y 608.509,Z 231.945,A -85,B 0,C 180,E1 -431.831,E2 -431.831} C_VEL
LIN {X 0,Y 608.477,Z 252.656,A -85,B 0,C 180,E1 -434.595,E2 -434.595} C_VEL
LIN {X 0,Y 608.441,Z 270.616,A -85,B 0,C 180,E1 -436.962,E2 -436.962} C_VEL
LIN {X 0,Y 608.571,Z 337.355,A -85,B 0,C 180,E1 -437.77,E2 -437.77} C_VEL
LIN {X 0,Y 608.526,Z 380.108,A -85,B 0,C 180,E1 -438.298,E2 -438.298} C_VEL
LIN {X 0,Y 608.517,Z 393.748,A -85,B 0,C 180,E1 -438.614,E2 -438.614} C_VEL
LIN {X 0,Y 608.509,Z 405.819,A -85,B 0,C 180,E1 -439.027,E2 -439.027} C_VEL
LIN {X 0,Y 608.494,Z 418.212,A -85,B 0,C 180,E1 -439.603,E2 -439.603} C_VEL
LIN {X 0,Y 608.506,Z 429.479,A -85,B 0,C 180,E1 -440.276,E2 -440.276} C_VEL
LIN {X 0,Y 608.474,Z 439.65,A -85,B 0,C 180,E1 -441.03,E2 -441.03} C_VEL
LIN {X 0,Y 608.464,Z 448.79,A -85,B 0,C 180,E1 -441.866,E2 -441.866} C_VEL
LIN {X 0,Y 608.466,Z 457.692,A -85,B 0,C 180,E1 -442.868,E2 -442.868} C_VEL
LIN {X 0,Y 608.443,Z 464.851,A -85,B 0,C 180,E1 -443.867,E2 -443.867} C_VEL
LIN {X 0,Y 608.463,Z 469.681,A -85,B 0,C 180,E1 -444.698,E2 -444.698} C_VEL
LIN {X 0,Y 608.439,Z 474.371,A -85,B 0,C 180,E1 -445.694,E2 -445.694} C_VEL
LIN {X 0,Y 608.424,Z 477.956,A -85,B 0,C 180,E1 -446.689,E2 -446.689} C_VEL
LIN {X 0,Y 608.425,Z 479.809,A -85,B 0,C 180,E1 -447.352,E2 -447.352} C_VEL
LIN {X 0,Y 608.444,Z 481.201,A -85,B 0,C 180,E1 -448.014,E2 -448.014} C_VEL
LIN {X 0,Y 608.439,Z 482.783,A -85,B 0,C 180,E1 -449.338,E2 -449.338} C_VEL
LIN {X 0,Y 608.434,Z 483,A -85,B 0,C 180,E1 -450,E2 -450} C_VEL
LIN {X 0,Y 608.448,Z 482.184,A -85,B 0,C 180,E1 -451.324,E2 -451.324} C_VEL
LIN {X 0,Y 608.444,Z 481.201,A -85,B 0,C 180,E1 -451.986,E2 -451.986} C_VEL
LIN {X 0,Y 608.425,Z 479.809,A -85,B 0,C 180,E1 -452.648,E2 -452.648} C_VEL
LIN {X 0,Y 608.449,Z 476.896,A -85,B 0,C 180,E1 -453.642,E2 -453.642} C_VEL
LIN {X 0,Y 608.432,Z 472.95,A -85,B 0,C 180,E1 -454.638,E2 -454.638} C_VEL
LIN {X 0,Y 608.437,Z 466.877,A -85,B 0,C 180,E1 -455.801,E2 -455.801} C_VEL
LIN {X 0,Y 608.463,Z 460.236,A -85,B 0,C 180,E1 -456.799,E2 -456.799} C_VEL
LIN {X 0,Y 608.456,Z 451.991,A -85,B 0,C 180,E1 -457.8,E2 -457.8} C_VEL
LIN {X 0,Y 608.472,Z 443.538,A -85,B 0,C 180,E1 -458.636,E2 -458.636} C_VEL
LIN {X 0,Y 608.479,Z 433.094,A -85,B 0,C 180,E1 -459.473,E2 -459.473} C_VEL
LIN {X 0,Y 608.498,Z 422.76,A -85,B 0,C 180,E1 -460.144,E2 -460.144} C_VEL
LIN {X 0,Y 608.517,Z 411.61,A -85,B 0,C 180,E1 -460.724,E2 -460.724} C_VEL
LIN {X 0,Y 608.517,Z 399.912,A -85,B 0,C 180,E1 -461.192,E2 -461.192} C_VEL
LIN {X 0,Y 608.53,Z 387.278,A -85,B 0,C 180,E1 -461.555,E2 -461.555} C_VEL
LIN {X 0,Y 608.534,Z 374.62,A -85,B 0,C 180,E1 -461.787,E2 -461.787} C_VEL
LIN {X 0,Y 608.496,Z 271.168,A -85,B 0,C 180,E1 -463.016,E2 -463.016} C_VEL
LIN {X 0,Y 608.444,Z 270.13,A -85,B 0,C 180,E1 -463.102,E2 -463.102} C_VEL
LIN {X 0,Y 608.495,Z 250.066,A -85,B 0,C 180,E1 -465.748,E2 -465.748} C_VEL
LIN {X 0,Y 608.514,Z 229.536,A -85,B 0,C 180,E1 -468.494,E2 -468.494} C_VEL
LIN {X 0,Y 608.54,Z 209.939,A -85,B 0,C 180,E1 -471.155,E2 -471.155} C_VEL
LIN {X 0,Y 608.404,Z 198.695,A -85,B 0,C 180,E1 -472.716,E2 -472.716} C_VEL
LIN {X 0,Y 608.399,Z 198.696,A -85,B 0,C 180,E1 -475.303,E2 -475.303} C_VEL
LIN {X 0,Y 608.404,Z 198.697,A -85,B 0,C 180,E1 -478.268,E2 -478.268} C_VEL
LIN {X 0,Y 608.401,Z 198.694,A -85,B 0,C 180,E1 -480.548,E2 -480.548} C_VEL
LIN {X 0,Y 608.406,Z 198.693,A -85,B 0,C 180,E1 -482.882,E2 -482.882} C_VEL
LIN {X 0,Y 608.409,Z 198.695,A -85,B 0,C 180,E1 -485.279,E2 -485.279} C_VEL
LIN {X 0,Y 608.408,Z 198.696,A -85,B 0,C 180,E1 -488.231,E2 -488.231} C_VEL
LIN {X 0,Y 608.404,Z 198.695,A -85,B 0,C 180,E1 -490.322,E2 -490.322} C_VEL
LIN {X 0,Y 608.383,Z 198.696,A -85,B 0,C 180,E1 -492.965,E2 -492.965} C_VEL
LIN {X 0,Y 608.446,Z 198.699,A -85,B 0,C 180,E1 -495.736,E2 -495.736} C_VEL
LIN {X 0,Y 608.451,Z 198.694,A -85,B 0,C 180,E1 -497.936,E2 -497.936} C_VEL
LIN {X 0,Y 608.396,Z 198.694,A -85,B 0,C 180,E1 -500.553,E2 -500.553} C_VEL
LIN {X 0,Y 608.389,Z 198.697,A -85,B 0,C 180,E1 -503.078,E2 -503.078} C_VEL
LIN {X 0,Y 608.434,Z 198.697,A -85,B 0,C 180,E1 -505.526,E2 -505.526} C_VEL
LIN {X 0,Y 608.448,Z 198.695,A -85,B 0,C 180,E1 -507.902,E2 -507.902} C_VEL
LIN {X 0,Y 608.416,Z 198.694,A -85,B 0,C 180,E1 -510.215,E2 -510.215} C_VEL
LIN {X 0,Y 608.398,Z 198.694,A -85,B 0,C 180,E1 -512.805,E2 -512.805} C_VEL
LIN {X 0,Y 608.425,Z 198.698,A -85,B 0,C 180,E1 -515.425,E2 -515.425} C_VEL
LIN {X 0,Y 608.416,Z 198.693,A -85,B 0,C 180,E1 -518.304,E2 -518.304} C_VEL
LIN {X 0,Y 608.394,Z 198.695,A -85,B 0,C 180,E1 -520.425,E2 -520.425} C_VEL
LIN {X 0,Y 608.417,Z 198.696,A -85,B 0,C 180,E1 -523.212,E2 -523.212} C_VEL
LIN {X 0,Y 608.421,Z 198.695,A -85,B 0,C 180,E1 -525.996,E2 -525.996} C_VEL
LIN {X 0,Y 608.417,Z 198.695,A -85,B 0,C 180,E1 -527.996,E2 -527.996} C_VEL
LIN {X 0,Y 608.409,Z 198.696,A -85,B 0,C 180,E1 -530.019,E2 -530.019} C_VEL
LIN {X 0,Y 608.394,Z 198.695,A -85,B 0,C 180,E1 -532.696,E2 -532.696} C_VEL
LIN {X 0,Y 608.443,Z 198.696,A -85,B 0,C 180,E1 -535.359,E2 -535.359} C_VEL
LIN {X 0,Y 608.404,Z 198.696,A -85,B 0,C 180,E1 -538.01,E2 -538.01} C_VEL
LIN {X 0,Y 608.427,Z 198.693,A -85,B 0,C 180,E1 -539.996,E2 -539.996} C_VEL
LIN {X 0,Y 608.409,Z 198.693,A -85,B 0,C 180,E1 -542.644,E2 -542.644} C_VEL
LIN {X 0,Y 608.44,Z 198.696,A -85,B 0,C 180,E1 -545.298,E2 -545.298} C_VEL
LIN {X 0,Y 608.401,Z 198.696,A -85,B 0,C 180,E1 -547.964,E2 -547.964} C_VEL
LIN {X 0,Y 608.43,Z 198.696,A -85,B 0,C 180,E1 -549.408,E2 -549.408} C_VEL
LIN {X 0,Y 607.738,Z 198.779,A -85,B 0,C 180,E1 -549.96,E2 -549.96} C_VEL
LIN {X 0,Y 604.883,Z 199.134,A -85,B 0,C 180,E1 -550.857,E2 -550.857} C_VEL
LIN {X 0,Y 602.481,Z 199.44,A -85,B 0,C 180,E1 -551.579,E2 -551.579} C_VEL
LIN {X 0,Y 601.442,Z 199.562,A -85,B 0,C 180,E1 -552.135,E2 -552.135} C_VEL
LIN {X 0,Y 601.352,Z 199.572,A -85,B 0,C 180,E1 -552.324,E2 -552.324} C_VEL
LIN {X 0,Y 601.365,Z 199.572,A -85,B 0,C 180,E1 -554.894,E2 -554.894} C_VEL
LIN {X 0,Y 601.361,Z 199.577,A -85,B 0,C 180,E1 -557.684,E2 -557.684} C_VEL
LIN {X 0,Y 601.364,Z 199.574,A -85,B 0,C 180,E1 -559.806,E2 -559.806} C_VEL
LIN {X 0,Y 601.368,Z 199.57,A -85,B 0,C 180,E1 -562.679,E2 -562.679} C_VEL
LIN {X 0,Y 601.401,Z 199.572,A -85,B 0,C 180,E1 -565.613,E2 -565.613} C_VEL
LIN {X 0,Y 601.353,Z 199.574,A -85,B 0,C 180,E1 -567.865,E2 -567.865} C_VEL
LIN {X 0,Y 601.36,Z 199.571,A -85,B 0,C 180,E1 -570.161,E2 -570.161} C_VEL
LIN {X 0,Y 601.367,Z 199.571,A -85,B 0,C 180,E1 -572.709,E2 -572.709} C_VEL
LIN {X 0,Y 601.354,Z 199.578,A -85,B 0,C 180,E1 -575.108,E2 -575.108} C_VEL
LIN {X 0,Y 601.394,Z 199.576,A -85,B 0,C 180,E1 -577.415,E2 -577.415} C_VEL
LIN {X 0,Y 601.364,Z 199.571,A -85,B 0,C 180,E1 -579.991,E2 -579.991} C_VEL
LIN {X 0,Y 601.362,Z 199.572,A -85,B 0,C 180,E1 -582.666,E2 -582.666} C_VEL
LIN {X 0,Y 601.373,Z 199.576,A -85,B 0,C 180,E1 -585.478,E2 -585.478} C_VEL
LIN {X 0,Y 601.366,Z 199.57,A -85,B 0,C 180,E1 -588.231,E2 -588.231} C_VEL
LIN {X 0,Y 601.389,Z 199.571,A -85,B 0,C 180,E1 -590.873,E2 -590.873} C_VEL
LIN {X 0,Y 601.39,Z 199.57,A -85,B 0,C 180,E1 -593.73,E2 -593.73} C_VEL
LIN {X 0,Y 601.36,Z 199.571,A -85,B 0,C 180,E1 -596.063,E2 -596.063} C_VEL
LIN {X 0,Y 601.384,Z 199.569,A -85,B 0,C 180,E1 -598.538,E2 -598.538} C_VEL
LIN {X 0,Y 601.402,Z 199.573,A -85,B 0,C 180,E1 -601.372,E2 -601.372} C_VEL
LIN {X 0,Y 601.355,Z 199.575,A -85,B 0,C 180,E1 -603.635,E2 -603.635} C_VEL
LIN {X 0,Y 601.368,Z 199.572,A -85,B 0,C 180,E1 -606.588,E2 -606.588} C_VEL
LIN {X 0,Y 601.394,Z 199.571,A -85,B 0,C 180,E1 -609.477,E2 -609.477} C_VEL
LIN {X 0,Y 601.342,Z 199.573,A -85,B 0,C 180,E1 -612.31,E2 -612.31} C_VEL
LIN {X 0,Y 601.363,Z 199.571,A -85,B 0,C 180,E1 -614.408,E2 -614.408} C_VEL
LIN {X 0,Y 601.377,Z 199.578,A -85,B 0,C 180,E1 -617.171,E2 -617.171} C_VEL
LIN {X 0,Y 601.394,Z 199.575,A -85,B 0,C 180,E1 -619.224,E2 -619.224} C_VEL
LIN {X 0,Y 601.373,Z 199.569,A -85,B 0,C 180,E1 -621.938,E2 -621.938} C_VEL
LIN {X 0,Y 601.346,Z 199.572,A -85,B 0,C 180,E1 -623.962,E2 -623.962} C_VEL
LIN {X 0,Y 601.392,Z 199.571,A -85,B 0,C 180,E1 -626.65,E2 -626.65} C_VEL
LIN {X 0,Y 601.412,Z 199.57,A -85,B 0,C 180,E1 -629.33,E2 -629.33} C_VEL
LIN {X 0,Y 601.354,Z 199.571,A -85,B 0,C 180,E1 -632.009,E2 -632.009} C_VEL
LIN {X 0,Y 601.38,Z 199.573,A -85,B 0,C 180,E1 -634.692,E2 -634.692} C_VEL
LIN {X 0,Y 601.402,Z 199.57,A -85,B 0,C 180,E1 -637.385,E2 -637.385} C_VEL
LIN {X 0,Y 601.371,Z 199.57,A -85,B 0,C 180,E1 -640.096,E2 -640.096} C_VEL
LIN {X 0,Y 601.356,Z 199.572,A -85,B 0,C 180,E1 -642.143,E2 -642.143} C_VEL
LIN {X 0,Y 601.371,Z 199.626,A -85,B 0,C 180,E1 -644.249,E2 -644.249} C_VEL
LIN {X 0,Y 601.433,Z 213.458,A -85,B 0,C 180,E1 -646.648,E2 -646.648} C_VEL
LIN {X 0,Y 601.4,Z 228.822,A -85,B 0,C 180,E1 -649.276,E2 -649.276} C_VEL
LIN {X 0,Y 601.363,Z 232.364,A -85,B 0,C 180,E1 -649.877,E2 -649.877} C_VEL
LIN {X 0,Y 601.656,Z 237.586,A -85,B 0,C 180,E1 -649.956,E2 -649.956} C_VEL
LIN {X 0,Y 601.579,Z 339.131,A -85,B 0,C 180,E1 -651.187,E2 -651.187} C_VEL
LIN {X 0,Y 601.555,Z 352.135,A -85,B 0,C 180,E1 -651.48,E2 -651.48} C_VEL
LIN {X 0,Y 601.545,Z 364.903,A -85,B 0,C 180,E1 -651.908,E2 -651.908} C_VEL
LIN {X 0,Y 601.511,Z 375.966,A -85,B 0,C 180,E1 -652.407,E2 -652.407} C_VEL
LIN {X 0,Y 601.449,Z 387.052,A -85,B 0,C 180,E1 -653.044,E2 -653.044} C_VEL
LIN {X 0,Y 601.466,Z 398.348,A -85,B 0,C 180,E1 -653.864,E2 -653.864} C_VEL
LIN {X 0,Y 601.428,Z 407.834,A -85,B 0,C 180,E1 -654.716,E2 -654.716} C_VEL
LIN {X 0,Y 601.384,Z 417.048,A -85,B 0,C 180,E1 -655.748,E2 -655.748} C_VEL
LIN {X 0,Y 601.357,Z 424.197,A -85,B 0,C 180,E1 -656.739,E2 -656.739} C_VEL
LIN {X 0,Y 601.343,Z 430.664,A -85,B 0,C 180,E1 -657.87,E2 -657.87} C_VEL
LIN {X 0,Y 601.328,Z 435.824,A -85,B 0,C 180,E1 -659.064,E2 -659.064} C_VEL
LIN {X 0,Y 601.355,Z 439.288,A -85,B 0,C 180,E1 -660.167,E2 -660.167} C_VEL
LIN {X 0,Y 601.353,Z 441.887,A -85,B 0,C 180,E1 -661.457,E2 -661.457} C_VEL
LIN {X 0,Y 601.322,Z 442.929,A -85,B 0,C 180,E1 -662.713,E2 -662.713} C_VEL
LIN {X 0,Y 601.31,Z 442.634,A -85,B 0,C 180,E1 -663.93,E2 -663.93} C_VEL
LIN {X 0,Y 601.319,Z 441.104,A -85,B 0,C 180,E1 -665.113,E2 -665.113} C_VEL
LIN {X 0,Y 601.342,Z 438.369,A -85,B 0,C 180,E1 -666.264,E2 -666.264} C_VEL
LIN {X 0,Y 601.367,Z 434.281,A -85,B 0,C 180,E1 -667.423,E2 -667.423} C_VEL
LIN {X 0,Y 601.337,Z 429.357,A -85,B 0,C 180,E1 -668.47,E2 -668.47} C_VEL
LIN {X 0,Y 601.378,Z 422.945,A -85,B 0,C 180,E1 -669.539,E2 -669.539} C_VEL
LIN {X 0,Y 601.412,Z 415.1,A -85,B 0,C 180,E1 -670.583,E2 -670.583} C_VEL
LIN {X 0,Y 601.418,Z 406.957,A -85,B 0,C 180,E1 -671.459,E2 -671.459} C_VEL
LIN {X 0,Y 601.454,Z 397.296,A -85,B 0,C 180,E1 -672.31,E2 -672.31} C_VEL
LIN {X 0,Y 601.495,Z 387.676,A -85,B 0,C 180,E1 -673.004,E2 -673.004} C_VEL
LIN {X 0,Y 601.511,Z 376.218,A -85,B 0,C 180,E1 -673.671,E2 -673.671} C_VEL
LIN {X 0,Y 601.522,Z 364.811,A -85,B 0,C 180,E1 -674.186,E2 -674.186} C_VEL
LIN {X 0,Y 601.557,Z 352.14,A -85,B 0,C 180,E1 -674.61,E2 -674.61} C_VEL
LIN {X 0,Y 601.604,Z 338.691,A -85,B 0,C 180,E1 -674.91,E2 -674.91} C_VEL
LIN {X 0,Y 601.634,Z 233.749,A -85,B 0,C 180,E1 -676.181,E2 -676.181} C_VEL
LIN {X 0,Y 601.426,Z 232.317,A -85,B 0,C 180,E1 -676.22,E2 -676.22} C_VEL
LIN {X 0,Y 601.451,Z 216.283,A -85,B 0,C 180,E1 -678.955,E2 -678.955} C_VEL
LIN {X 0,Y 601.476,Z 201.435,A -85,B 0,C 180,E1 -681.522,E2 -681.522} C_VEL
LIN {X 0,Y 601.413,Z 199.567,A -85,B 0,C 180,E1 -681.872,E2 -681.872} C_VEL
LIN {X 0,Y 601.414,Z 199.571,A -85,B 0,C 180,E1 -684.883,E2 -684.883} C_VEL
LIN {X 0,Y 601.395,Z 199.57,A -85,B 0,C 180,E1 -687.489,E2 -687.489} C_VEL
LIN {X 0,Y 601.409,Z 199.565,A -85,B 0,C 180,E1 -689.852,E2 -689.852} C_VEL
LIN {X 0,Y 601.446,Z 199.569,A -85,B 0,C 180,E1 -692.895,E2 -692.895} C_VEL
LIN {X 0,Y 601.414,Z 199.564,A -85,B 0,C 180,E1 -695.864,E2 -695.864} C_VEL
LIN {X 0,Y 601.388,Z 199.574,A -85,B 0,C 180,E1 -698.765,E2 -698.765} C_VEL
LIN {X 0,Y 601.368,Z 199.571,A -85,B 0,C 180,E1 -701.612,E2 -701.612} C_VEL
LIN {X 0,Y 601.398,Z 199.567,A -85,B 0,C 180,E1 -703.717,E2 -703.717} C_VEL
LIN {X 0,Y 601.403,Z 199.569,A -85,B 0,C 180,E1 -706.489,E2 -706.489} C_VEL
LIN {X 0,Y 601.398,Z 199.571,A -85,B 0,C 180,E1 -709.228,E2 -709.228} C_VEL
LIN {X 0,Y 601.408,Z 199.565,A -85,B 0,C 180,E1 -711.943,E2 -711.943} C_VEL
LIN {X 0,Y 601.426,Z 199.57,A -85,B 0,C 180,E1 -714.64,E2 -714.64} C_VEL
LIN {X 0,Y 601.404,Z 199.568,A -85,B 0,C 180,E1 -717.325,E2 -717.325} C_VEL
LIN {X 0,Y 601.408,Z 199.565,A -85,B 0,C 180,E1 -720.004,E2 -720.004} C_VEL
LIN {X 0,Y 601.441,Z 199.57,A -85,B 0,C 180,E1 -722.683,E2 -722.683} C_VEL
LIN {X 0,Y 601.387,Z 199.569,A -85,B 0,C 180,E1 -725.368,E2 -725.368} C_VEL
LIN {X 0,Y 601.391,Z 199.568,A -85,B 0,C 180,E1 -728.065,E2 -728.065} C_VEL
LIN {X 0,Y 601.405,Z 199.57,A -85,B 0,C 180,E1 -731.01,E2 -731.01} C_VEL
LIN {X 0,Y 601.372,Z 199.569,A -85,B 0,C 180,E1 -733.52,E2 -733.52} C_VEL
LIN {X 0,Y 601.426,Z 199.568,A -85,B 0,C 180,E1 -736.29,E2 -736.29} C_VEL
LIN {X 0,Y 601.399,Z 199.568,A -85,B 0,C 180,E1 -739.102,E2 -739.102} C_VEL
LIN {X 0,Y 601.38,Z 199.569,A -85,B 0,C 180,E1 -741.243,E2 -741.243} C_VEL
LIN {X 0,Y 601.433,Z 199.566,A -85,B 0,C 180,E1 -744.144,E2 -744.144} C_VEL
LIN {X 0,Y 601.378,Z 199.57,A -85,B 0,C 180,E1 -747.117,E2 -747.117} C_VEL
LIN {X 0,Y 601.37,Z 199.57,A -85,B 0,C 180,E1 -749.398,E2 -749.398} C_VEL
LIN {X 0,Y 601.433,Z 199.572,A -85,B 0,C 180,E1 -752.518,E2 -752.518} C_VEL
LIN {X 0,Y 601.358,Z 199.572,A -85,B 0,C 180,E1 -755.109,E2 -755.109} C_VEL
LIN {X 0,Y 601.38,Z 199.568,A -85,B 0,C 180,E1 -757.425,E2 -757.425} C_VEL
LIN {X 0,Y 601.391,Z 199.571,A -85,B 0,C 180,E1 -759.999,E2 -759.999} C_VEL
LIN {X 0,Y 601.375,Z 199.574,A -85,B 0,C 180,E1 -762.675,E2 -762.675} C_VEL
LIN {X 0,Y 601.366,Z 199.57,A -85,B 0,C 180,E1 -765.478,E2 -765.478} C_VEL
LIN {X 0,Y 601.401,Z 199.575,A -85,B 0,C 180,E1 -768.411,E2 -768.411} C_VEL
LIN {X 0,Y 601.376,Z 199.571,A -85,B 0,C 180,E1 -770.872,E2 -770.872} C_VEL
LIN {X 0,Y 601.382,Z 199.571,A -85,B 0,C 180,E1 -773.744,E2 -773.744} C_VEL
LIN {X 0,Y 601.379,Z 199.572,A -85,B 0,C 180,E1 -776.685,E2 -776.685} C_VEL
LIN {X 0,Y 601.377,Z 199.569,A -85,B 0,C 180,E1 -779.057,E2 -779.057} C_VEL
LIN {X 0,Y 601.35,Z 199.573,A -85,B 0,C 180,E1 -781.37,E2 -781.37} C_VEL
LIN {X 0,Y 601.399,Z 199.574,A -85,B 0,C 180,E1 -784.382,E2 -784.382} C_VEL
LIN {X 0,Y 601.374,Z 199.573,A -85,B 0,C 180,E1 -787.112,E2 -787.112} C_VEL
LIN {X 0,Y 601.653,Z 204.807,A -85,B 0,C 180,E1 -787.877,E2 -787.877} C_VEL
LIN {X 0,Y 601.596,Z 224.178,A -85,B 0,C 180,E1 -790.553,E2 -790.553} C_VEL
LIN {X 0,Y 601.522,Z 245.656,A -85,B 0,C 180,E1 -793.47,E2 -793.47} C_VEL
LIN {X 0,Y 601.481,Z 267.08,A -85,B 0,C 180,E1 -796.338,E2 -796.338} C_VEL
LIN {X 0,Y 601.417,Z 270.616,A -85,B 0,C 180,E1 -796.807,E2 -796.807} C_VEL
LIN {X 0,Y 601.658,Z 274.752,A -85,B 0,C 180,E1 -796.877,E2 -796.877} C_VEL
LIN {X 0,Y 601.605,Z 378.966,A -85,B 0,C 180,E1 -798.14,E2 -798.14} C_VEL
LIN {X 0,Y 601.566,Z 392.23,A -85,B 0,C 180,E1 -798.438,E2 -798.438} C_VEL
LIN {X 0,Y 601.544,Z 403.928,A -85,B 0,C 180,E1 -798.826,E2 -798.826} C_VEL
LIN {X 0,Y 601.524,Z 416.639,A -85,B 0,C 180,E1 -799.396,E2 -799.396} C_VEL
LIN {X 0,Y 601.485,Z 428.204,A -85,B 0,C 180,E1 -800.076,E2 -800.076} C_VEL
LIN {X 0,Y 601.444,Z 438.599,A -85,B 0,C 180,E1 -800.839,E2 -800.839} C_VEL
LIN {X 0,Y 601.429,Z 447.115,A -85,B 0,C 180,E1 -801.601,E2 -801.601} C_VEL
LIN {X 0,Y 601.418,Z 454.962,A -85,B 0,C 180,E1 -802.446,E2 -802.446} C_VEL
LIN {X 0,Y 601.371,Z 462.229,A -85,B 0,C 180,E1 -803.399,E2 -803.399} C_VEL
LIN {X 0,Y 601.372,Z 467.867,A -85,B 0,C 180,E1 -804.299,E2 -804.299} C_VEL
LIN {X 0,Y 601.336,Z 472.951,A -85,B 0,C 180,E1 -805.307,E2 -805.307} C_VEL
LIN {X 0,Y 601.368,Z 476.896,A -85,B 0,C 180,E1 -806.315,E2 -806.315} C_VEL
LIN {X 0,Y 601.325,Z 479.809,A -85,B 0,C 180,E1 -807.321,E2 -807.321} C_VEL
LIN {X 0,Y 601.343,Z 481.202,A -85,B 0,C 180,E1 -807.991,E2 -807.991} C_VEL
LIN {X 0,Y 601.339,Z 482.784,A -85,B 0,C 180,E1 -809.33,E2 -809.33} C_VEL
LIN {X 0,Y 601.335,Z 483,A -85,B 0,C 180,E1 -810,E2 -810} C_VEL
LIN {X 0,Y 601.348,Z 482.184,A -85,B 0,C 180,E1 -811.339,E2 -811.339} C_VEL
LIN {X 0,Y 601.343,Z 481.202,A -85,B 0,C 180,E1 -812.009,E2 -812.009} C_VEL
LIN {X 0,Y 601.325,Z 479.809,A -85,B 0,C 180,E1 -812.68,E2 -812.68} C_VEL
LIN {X 0,Y 601.368,Z 476.896,A -85,B 0,C 180,E1 -813.685,E2 -813.685} C_VEL
LIN {X 0,Y 601.336,Z 472.95,A -85,B 0,C 180,E1 -814.693,E2 -814.693} C_VEL
LIN {X 0,Y 601.372,Z 466.878,A -85,B 0,C 180,E1 -815.869,E2 -815.869} C_VEL
LIN {X 0,Y 601.383,Z 460.237,A -85,B 0,C 180,E1 -816.88,E2 -816.88} C_VEL
LIN {X 0,Y 601.401,Z 451.991,A -85,B 0,C 180,E1 -817.892,E2 -817.892} C_VEL
LIN {X 0,Y 601.436,Z 443.539,A -85,B 0,C 180,E1 -818.737,E2 -818.737} C_VEL
LIN {X 0,Y 601.449,Z 433.096,A -85,B 0,C 180,E1 -819.585,E2 -819.585} C_VEL
LIN {X 0,Y 601.476,Z 422.762,A -85,B 0,C 180,E1 -820.264,E2 -820.264} C_VEL
LIN {X 0,Y 601.539,Z 410.6,A -85,B 0,C 180,E1 -820.896,E2 -820.896} C_VEL
LIN {X 0,Y 601.551,Z 398.225,A -85,B 0,C 180,E1 -821.379,E2 -821.379} C_VEL
LIN {X 0,Y 601.569,Z 385.449,A -85,B 0,C 180,E1 -821.733,E2 -821.733} C_VEL
LIN {X 0,Y 601.611,Z 373.105,A -85,B 0,C 180,E1 -821.946,E2 -821.946} C_VEL
LIN {X 0,Y 601.471,Z 271.168,A -85,B 0,C 180,E1 -823.17,E2 -823.17} C_VEL
LIN {X 0,Y 601.455,Z 270.13,A -85,B 0,C 180,E1 -823.257,E2 -823.257} C_VEL
LIN {X 0,Y 601.52,Z 248.772,A -85,B 0,C 180,E1 -826.11,E2 -826.11} C_VEL
LIN {X 0,Y 601.598,Z 226.766,A -85,B 0,C 180,E1 -829.093,E2 -829.093} C_VEL
LIN {X 0,Y 601.662,Z 206.055,A -85,B 0,C 180,E1 -831.949,E2 -831.949} C_VEL
LIN {X 0,Y 601.355,Z 199.583,A -85,B 0,C 180,E1 -832.866,E2 -832.866} C_VEL
LIN {X 0,Y 601.359,Z 199.572,A -85,B 0,C 180,E1 -834.88,E2 -834.88} C_VEL
LIN {X 0,Y 601.362,Z 199.574,A -85,B 0,C 180,E1 -837.351,E2 -837.351} C_VEL
LIN {X 0,Y 601.402,Z 199.571,A -85,B 0,C 180,E1 -840.165,E2 -840.165} C_VEL
LIN {X 0,Y 601.374,Z 199.569,A -85,B 0,C 180,E1 -842.707,E2 -842.707} C_VEL
LIN {X 0,Y 601.348,Z 199.573,A -85,B 0,C 180,E1 -845.104,E2 -845.104} C_VEL
LIN {X 0,Y 601.386,Z 199.572,A -85,B 0,C 180,E1 -847.422,E2 -847.422} C_VEL
LIN {X 0,Y 601.376,Z 199.575,A -85,B 0,C 180,E1 -849.997,E2 -849.997} C_VEL
LIN {X 0,Y 601.339,Z 199.574,A -85,B 0,C 180,E1 -852.581,E2 -852.581} C_VEL
LIN {X 0,Y 601.366,Z 199.57,A -85,B 0,C 180,E1 -854.528,E2 -854.528} C_VEL
LIN {X 0,Y 601.364,Z 199.574,A -85,B 0,C 180,E1 -857.324,E2 -857.324} C_VEL
LIN {X 0,Y 601.389,Z 199.573,A -85,B 0,C 180,E1 -860.001,E2 -860.001} C_VEL
LIN {X 0,Y 601.343,Z 199.573,A -85,B 0,C 180,E1 -862.628,E2 -862.628} C_VEL
LIN {X 0,Y 601.359,Z 199.572,A -85,B 0,C 180,E1 -865.062,E2 -865.062} C_VEL
LIN {X 0,Y 601.42,Z 199.57,A -85,B 0,C 180,E1 -867.481,E2 -867.481} C_VEL
LIN {X 0,Y 601.359,Z 199.571,A -85,B 0,C 180,E1 -870.601,E2 -870.601} C_VEL
LIN {X 0,Y 601.364,Z 199.571,A -85,B 0,C 180,E1 -872.882,E2 -872.882} C_VEL
LIN {X 0,Y 601.432,Z 199.569,A -85,B 0,C 180,E1 -875.856,E2 -875.856} C_VEL
LIN {X 0,Y 601.375,Z 199.573,A -85,B 0,C 180,E1 -878.037,E2 -878.037} C_VEL
LIN {X 0,Y 601.364,Z 199.572,A -85,B 0,C 180,E1 -880.186,E2 -880.186} C_VEL
LIN {X 0,Y 601.364,Z 199.572,A -85,B 0,C 180,E1 -883.009,E2 -883.009} C_VEL
LIN {X 0,Y 601.366,Z 199.575,A -85,B 0,C 180,E1 -885.924,E2 -885.924} C_VEL
LIN {X 0,Y 601.359,Z 199.571,A -85,B 0,C 180,E1 -888.537,E2 -888.537} C_VEL
LIN {X 0,Y 601.389,Z 199.573,A -85,B 0,C 180,E1 -891.258,E2 -891.258} C_VEL
LIN {X 0,Y 601.367,Z 199.574,A -85,B 0,C 180,E1 -893.959,E2 -893.959} C_VEL
LIN {X 0,Y 601.356,Z 199.575,A -85,B 0,C 180,E1 -895.975,E2 -895.975} C_VEL
LIN {X 0,Y 601.379,Z 199.572,A -85,B 0,C 180,E1 -897.987,E2 -897.987} C_VEL
LIN {X 0,Y 601.399,Z 199.569,A -85,B 0,C 180,E1 -899.996,E2 -899.996} C_VEL
LIN {X 0,Y 601.381,Z 199.568,A -85,B 0,C 180,E1 -902.675,E2 -902.675} C_VEL
LIN {X 0,Y 601.402,Z 199.574,A -85,B 0,C 180,E1 -905.36,E2 -905.36} C_VEL
LIN {X 0,Y 601.373,Z 199.571,A -85,B 0,C 180,E1 -908.057,E2 -908.057} C_VEL
LIN {X 0,Y 601.359,Z 199.572,A -85,B 0,C 180,E1 -910.773,E2 -910.773} C_VEL
LIN {X 0,Y 601.352,Z 199.572,A -85,B 0,C 180,E1 -912.324,E2 -912.324} C_VEL
LIN {X 0,Y 600.674,Z 199.659,A -85,B 0,C 180,E1 -912.883,E2 -912.883} C_VEL
LIN {X 0,Y 597.826,Z 200.016,A -85,B 0,C 180,E1 -913.791,E2 -913.791} C_VEL
LIN {X 0,Y 595.427,Z 200.315,A -85,B 0,C 180,E1 -914.521,E2 -914.521} C_VEL
LIN {X 0,Y 594.397,Z 200.443,A -85,B 0,C 180,E1 -915.084,E2 -915.084} C_VEL
LIN {X 0,Y 594.312,Z 200.452,A -85,B 0,C 180,E1 -915.275,E2 -915.275} C_VEL
LIN {X 0,Y 594.307,Z 200.452,A -85,B 0,C 180,E1 -917.901,E2 -917.901} C_VEL
LIN {X 0,Y 594.351,Z 200.445,A -85,B 0,C 180,E1 -920.772,E2 -920.772} C_VEL
LIN {X 0,Y 594.331,Z 200.451,A -85,B 0,C 180,E1 -923.701,E2 -923.701} C_VEL
LIN {X 0,Y 594.322,Z 200.449,A -85,B 0,C 180,E1 -926.013,E2 -926.013} C_VEL
LIN {X 0,Y 594.322,Z 200.448,A -85,B 0,C 180,E1 -928.224,E2 -928.224} C_VEL
LIN {X 0,Y 594.333,Z 200.447,A -85,B 0,C 180,E1 -930.556,E2 -930.556} C_VEL
LIN {X 0,Y 594.335,Z 200.45,A -85,B 0,C 180,E1 -932.946,E2 -932.946} C_VEL
LIN {X 0,Y 594.307,Z 200.459,A -85,B 0,C 180,E1 -935.405,E2 -935.405} C_VEL
LIN {X 0,Y 594.332,Z 200.448,A -85,B 0,C 180,E1 -937.937,E2 -937.937} C_VEL
LIN {X 0,Y 594.335,Z 200.449,A -85,B 0,C 180,E1 -940.819,E2 -940.819} C_VEL
LIN {X 0,Y 594.332,Z 200.448,A -85,B 0,C 180,E1 -943.837,E2 -943.837} C_VEL
LIN {X 0,Y 594.32,Z 200.45,A -85,B 0,C 180,E1 -946.698,E2 -946.698} C_VEL
LIN {X 0,Y 594.336,Z 200.453,A -85,B 0,C 180,E1 -949.432,E2 -949.432} C_VEL
LIN {X 0,Y 594.334,Z 200.446,A -85,B 0,C 180,E1 -952.388,E2 -952.388} C_VEL
LIN {X 0,Y 594.347,Z 200.447,A -85,B 0,C 180,E1 -954.666,E2 -954.666} C_VEL
LIN {X 0,Y 594.322,Z 200.456,A -85,B 0,C 180,E1 -957.085,E2 -957.085} C_VEL
LIN {X 0,Y 594.34,Z 200.448,A -85,B 0,C 180,E1 -959.666,E2 -959.666} C_VEL
LIN {X 0,Y 594.328,Z 200.448,A -85,B 0,C 180,E1 -962.538,E2 -962.538} C_VEL
LIN {X 0,Y 594.322,Z 200.452,A -85,B 0,C 180,E1 -964.805,E2 -964.805} C_VEL
LIN {X 0,Y 594.342,Z 200.454,A -85,B 0,C 180,E1 -967.252,E2 -967.252} C_VEL
LIN {X 0,Y 594.323,Z 200.448,A -85,B 0,C 180,E1 -969.945,E2 -969.945} C_VEL
LIN {X 0,Y 594.334,Z 200.451,A -85,B 0,C 180,E1 -972.805,E2 -972.805} C_VEL
LIN {X 0,Y 594.342,Z 200.446,A -85,B 0,C 180,E1 -975.815,E2 -975.815} C_VEL
LIN {X 0,Y 594.399,Z 200.445,A -85,B 0,C 180,E1 -978.885,E2 -978.885} C_VEL
LIN {X 0,Y 594.351,Z 200.444,A -85,B 0,C 180,E1 -981.843,E2 -981.843} C_VEL
LIN {X 0,Y 594.306,Z 200.45,A -85,B 0,C 180,E1 -983.891,E2 -983.891} C_VEL
LIN {X 0,Y 594.341,Z 200.448,A -85,B 0,C 180,E1 -986.61,E2 -986.61} C_VEL
LIN {X 0,Y 594.38,Z 200.446,A -85,B 0,C 180,E1 -989.322,E2 -989.322} C_VEL
LIN {X 0,Y 594.325,Z 200.447,A -85,B 0,C 180,E1 -992.033,E2 -992.033} C_VEL
LIN {X 0,Y 594.349,Z 200.45,A -85,B 0,C 180,E1 -994.748,E2 -994.748} C_VEL
LIN {X 0,Y 594.36,Z 200.446,A -85,B 0,C 180,E1 -997.473,E2 -997.473} C_VEL
LIN {X 0,Y 594.337,Z 200.447,A -85,B 0,C 180,E1 -1000.217,E2 -1000.217} C_VEL
LIN {X 0,Y 594.332,Z 200.448,A -85,B 0,C 180,E1 -1002.289,E2 -1002.289} C_VEL
LIN {X 0,Y 594.37,Z 200.619,A -85,B 0,C 180,E1 -1004.195,E2 -1004.195} C_VEL
LIN {X 0,Y 594.438,Z 216.136,A -85,B 0,C 180,E1 -1006.916,E2 -1006.916} C_VEL
LIN {X 0,Y 594.345,Z 232.22,A -85,B 0,C 180,E1 -1009.694,E2 -1009.694} C_VEL
LIN {X 0,Y 594.581,Z 233.962,A -85,B 0,C 180,E1 -1009.753,E2 -1009.753} C_VEL
LIN {X 0,Y 594.659,Z 328.184,A -85,B 0,C 180,E1 -1010.898,E2 -1010.898} C_VEL
LIN {X 0,Y 594.644,Z 343.686,A -85,B 0,C 180,E1 -1011.133,E2 -1011.133} C_VEL
LIN {X 0,Y 594.601,Z 355.969,A -85,B 0,C 180,E1 -1011.457,E2 -1011.457} C_VEL
LIN {X 0,Y 594.54,Z 368.017,A -85,B 0,C 180,E1 -1011.906,E2 -1011.906} C_VEL
LIN {X 0,Y 594.5,Z 380.594,A -85,B 0,C 180,E1 -1012.532,E2 -1012.532} C_VEL
LIN {X 0,Y 594.448,Z 391.647,A -85,B 0,C 180,E1 -1013.239,E2 -1013.239} C_VEL
LIN {X 0,Y 594.392,Z 402.076,A -85,B 0,C 180,E1 -1014.074,E2 -1014.074} C_VEL
LIN {X 0,Y 594.357,Z 411.529,A -85,B 0,C 180,E1 -1015.006,E2 -1015.006} C_VEL
LIN {X 0,Y 594.299,Z 419.789,A -85,B 0,C 180,E1 -1016.021,E2 -1016.021} C_VEL
LIN {X 0,Y 594.286,Z 426.746,A -85,B 0,C 180,E1 -1017.083,E2 -1017.083} C_VEL
LIN {X 0,Y 594.286,Z 432.663,A -85,B 0,C 180,E1 -1018.231,E2 -1018.231} C_VEL
LIN {X 0,Y 594.258,Z 437.138,A -85,B 0,C 180,E1 -1019.392,E2 -1019.392} C_VEL
LIN {X 0,Y 594.252,Z 440.316,A -85,B 0,C 180,E1 -1020.566,E2 -1020.566} C_VEL
LIN {X 0,Y 594.233,Z 442.12,A -85,B 0,C 180,E1 -1021.633,E2 -1021.633} C_VEL
LIN {X 0,Y 594.214,Z 442.986,A -85,B 0,C 180,E1 -1022.959,E2 -1022.959} C_VEL
LIN {X 0,Y 594.227,Z 442.494,A -85,B 0,C 180,E1 -1024.128,E2 -1024.128} C_VEL
LIN {X 0,Y 594.226,Z 440.542,A -85,B 0,C 180,E1 -1025.416,E2 -1025.416} C_VEL
LIN {X 0,Y 594.26,Z 437.822,A -85,B 0,C 180,E1 -1026.478,E2 -1026.478} C_VEL
LIN {X 0,Y 594.258,Z 433.749,A -85,B 0,C 180,E1 -1027.603,E2 -1027.603} C_VEL
LIN {X 0,Y 594.278,Z 427.879,A -85,B 0,C 180,E1 -1028.812,E2 -1028.812} C_VEL
LIN {X 0,Y 594.331,Z 420.745,A -85,B 0,C 180,E1 -1029.937,E2 -1029.937} C_VEL
LIN {X 0,Y 594.349,Z 412.864,A -85,B 0,C 180,E1 -1030.931,E2 -1030.931} C_VEL
LIN {X 0,Y 594.403,Z 403.829,A -85,B 0,C 180,E1 -1031.86,E2 -1031.86} C_VEL
LIN {X 0,Y 594.431,Z 394.771,A -85,B 0,C 180,E1 -1032.62,E2 -1032.62} C_VEL
LIN {X 0,Y 594.487,Z 383.321,A -85,B 0,C 180,E1 -1033.397,E2 -1033.397} C_VEL
LIN {X 0,Y 594.56,Z 371.17,A -85,B 0,C 180,E1 -1034.045,E2 -1034.045} C_VEL
LIN {X 0,Y 594.598,Z 359.808,A -85,B 0,C 180,E1 -1034.506,E2 -1034.506} C_VEL
LIN {X 0,Y 594.624,Z 346.513,A -85,B 0,C 180,E1 -1034.892,E2 -1034.892} C_VEL
LIN {X 0,Y 594.68,Z 333.806,A -85,B 0,C 180,E1 -1035.122,E2 -1035.122} C_VEL
LIN {X 0,Y 594.65,Z 234.193,A -85,B 0,C 180,E1 -1036.332,E2 -1036.332} C_VEL
LIN {X 0,Y 594.372,Z 232.337,A -85,B 0,C 180,E1 -1036.375,E2 -1036.375} C_VEL
LIN {X 0,Y 594.442,Z 216.162,A -85,B 0,C 180,E1 -1039.169,E2 -1039.169} C_VEL
LIN {X 0,Y 594.459,Z 202.038,A -85,B 0,C 180,E1 -1041.642,E2 -1041.642} C_VEL
LIN {X 0,Y 594.358,Z 200.447,A -85,B 0,C 180,E1 -1041.957,E2 -1041.957} C_VEL
LIN {X 0,Y 594.362,Z 200.447,A -85,B 0,C 180,E1 -1044.673,E2 -1044.673} C_VEL
LIN {X 0,Y 594.346,Z 200.455,A -85,B 0,C 180,E1 -1047.091,E2 -1047.091} C_VEL
LIN {X 0,Y 594.363,Z 200.444,A -85,B 0,C 180,E1 -1049.673,E2 -1049.673} C_VEL
LIN {X 0,Y 594.363,Z 200.446,A -85,B 0,C 180,E1 -1052.545,E2 -1052.545} C_VEL
LIN {X 0,Y 594.355,Z 200.451,A -85,B 0,C 180,E1 -1054.812,E2 -1054.812} C_VEL
LIN {X 0,Y 594.336,Z 200.451,A -85,B 0,C 180,E1 -1057.268,E2 -1057.268} C_VEL
LIN {X 0,Y 594.347,Z 200.445,A -85,B 0,C 180,E1 -1059.951,E2 -1059.951} C_VEL
LIN {X 0,Y 594.367,Z 200.451,A -85,B 0,C 180,E1 -1062.811,E2 -1062.811} C_VEL
LIN {X 0,Y 594.351,Z 200.444,A -85,B 0,C 180,E1 -1065.835,E2 -1065.835} C_VEL
LIN {X 0,Y 594.418,Z 200.446,A -85,B 0,C 180,E1 -1068.905,E2 -1068.905} C_VEL
LIN {X 0,Y 594.355,Z 200.443,A -85,B 0,C 180,E1 -1071.847,E2 -1071.847} C_VEL
LIN {X 0,Y 594.385,Z 200.446,A -85,B 0,C 180,E1 -1074.576,E2 -1074.576} C_VEL
LIN {X 0,Y 594.374,Z 200.444,A -85,B 0,C 180,E1 -1077.293,E2 -1077.293} C_VEL
LIN {X 0,Y 594.379,Z 200.441,A -85,B 0,C 180,E1 -1080.004,E2 -1080.004} C_VEL
LIN {X 0,Y 594.402,Z 200.448,A -85,B 0,C 180,E1 -1082.714,E2 -1082.714} C_VEL
LIN {X 0,Y 594.353,Z 200.444,A -85,B 0,C 180,E1 -1085.432,E2 -1085.432} C_VEL
LIN {X 0,Y 594.334,Z 200.447,A -85,B 0,C 180,E1 -1087.477,E2 -1087.477} C_VEL
LIN {X 0,Y 594.325,Z 200.447,A -85,B 0,C 180,E1 -1089.533,E2 -1089.533} C_VEL
LIN {X 0,Y 594.37,Z 200.446,A -85,B 0,C 180,E1 -1092.292,E2 -1092.292} C_VEL
LIN {X 0,Y 594.352,Z 200.447,A -85,B 0,C 180,E1 -1095.082,E2 -1095.082} C_VEL
LIN {X 0,Y 594.364,Z 200.444,A -85,B 0,C 180,E1 -1097.197,E2 -1097.197} C_VEL
LIN {X 0,Y 594.354,Z 200.446,A -85,B 0,C 180,E1 -1100.057,E2 -1100.057} C_VEL
LIN {X 0,Y 594.342,Z 200.449,A -85,B 0,C 180,E1 -1102.971,E2 -1102.971} C_VEL
LIN {X 0,Y 594.315,Z 200.45,A -85,B 0,C 180,E1 -1105.198,E2 -1105.198} C_VEL
LIN {X 0,Y 594.34,Z 200.445,A -85,B 0,C 180,E1 -1107.521,E2 -1107.521} C_VEL
LIN {X 0,Y 594.343,Z 200.446,A -85,B 0,C 180,E1 -1109.781,E2 -1109.781} C_VEL
LIN {X 0,Y 594.359,Z 200.448,A -85,B 0,C 180,E1 -1112.15,E2 -1112.15} C_VEL
LIN {X 0,Y 594.352,Z 200.452,A -85,B 0,C 180,E1 -1114.584,E2 -1114.584} C_VEL
LIN {X 0,Y 594.349,Z 200.445,A -85,B 0,C 180,E1 -1117.605,E2 -1117.605} C_VEL
LIN {X 0,Y 594.336,Z 200.447,A -85,B 0,C 180,E1 -1119.772,E2 -1119.772} C_VEL
LIN {X 0,Y 594.346,Z 200.455,A -85,B 0,C 180,E1 -1122.379,E2 -1122.379} C_VEL
LIN {X 0,Y 594.314,Z 200.449,A -85,B 0,C 180,E1 -1125.198,E2 -1125.198} C_VEL
LIN {X 0,Y 594.361,Z 200.451,A -85,B 0,C 180,E1 -1128.156,E2 -1128.156} C_VEL
LIN {X 0,Y 594.323,Z 200.448,A -85,B 0,C 180,E1 -1131.192,E2 -1131.192} C_VEL
LIN {X 0,Y 594.336,Z 200.449,A -85,B 0,C 180,E1 -1133.756,E2 -1133.756} C_VEL
LIN {X 0,Y 594.351,Z 200.455,A -85,B 0,C 180,E1 -1136.238,E2 -1136.238} C_VEL
LIN {X 0,Y 594.337,Z 200.45,A -85,B 0,C 180,E1 -1138.649,E2 -1138.649} C_VEL
LIN {X 0,Y 594.331,Z 200.447,A -85,B 0,C 180,E1 -1141.053,E2 -1141.053} C_VEL
LIN {X 0,Y 594.335,Z 200.454,A -85,B 0,C 180,E1 -1143.989,E2 -1143.989} C_VEL
LIN {X 0,Y 594.332,Z 200.452,A -85,B 0,C 180,E1 -1146.848,E2 -1146.848} C_VEL
LIN {X 0,Y 594.338,Z 200.555,A -85,B 0,C 180,E1 -1146.986,E2 -1146.986} C_VEL
LIN {X 0,Y 594.739,Z 205.052,A -85,B 0,C 180,E1 -1147.64,E2 -1147.64} C_VEL
LIN {X 0,Y 594.65,Z 225.472,A -85,B 0,C 180,E1 -1150.496,E2 -1150.496} C_VEL
LIN {X 0,Y 594.548,Z 247.478,A -85,B 0,C 180,E1 -1153.519,E2 -1153.519} C_VEL
LIN {X 0,Y 594.425,Z 269.483,A -85,B 0,C 180,E1 -1156.497,E2 -1156.497} C_VEL
LIN {X 0,Y 594.436,Z 270.616,A -85,B 0,C 180,E1 -1156.649,E2 -1156.649} C_VEL
LIN {X 0,Y 594.739,Z 274.752,A -85,B 0,C 180,E1 -1156.721,E2 -1156.721} C_VEL
LIN {X 0,Y 594.657,Z 378.966,A -85,B 0,C 180,E1 -1157.999,E2 -1157.999} C_VEL
LIN {X 0,Y 594.629,Z 392.231,A -85,B 0,C 180,E1 -1158.301,E2 -1158.301} C_VEL
LIN {X 0,Y 594.576,Z 404.515,A -85,B 0,C 180,E1 -1158.716,E2 -1158.716} C_VEL
LIN {X 0,Y 594.528,Z 416.638,A -85,B 0,C 180,E1 -1159.27,E2 -1159.27} C_VEL
LIN {X 0,Y 594.473,Z 428.205,A -85,B 0,C 180,E1 -1159.958,E2 -1159.958} C_VEL
LIN {X 0,Y 594.414,Z 438.601,A -85,B 0,C 180,E1 -1160.73,E2 -1160.73} C_VEL
LIN {X 0,Y 594.366,Z 447.115,A -85,B 0,C 180,E1 -1161.501,E2 -1161.501} C_VEL
LIN {X 0,Y 594.348,Z 454.962,A -85,B 0,C 180,E1 -1162.356,E2 -1162.356} C_VEL
LIN {X 0,Y 594.283,Z 462.82,A -85,B 0,C 180,E1 -1163.409,E2 -1163.409} C_VEL
LIN {X 0,Y 594.289,Z 469.681,A -85,B 0,C 180,E1 -1164.571,E2 -1164.571} C_VEL
LIN {X 0,Y 594.271,Z 474.372,A -85,B 0,C 180,E1 -1165.591,E2 -1165.591} C_VEL
LIN {X 0,Y 594.267,Z 477.957,A -85,B 0,C 180,E1 -1166.61,E2 -1166.61} C_VEL
LIN {X 0,Y 594.226,Z 479.809,A -85,B 0,C 180,E1 -1167.289,E2 -1167.289} C_VEL
LIN {X 0,Y 594.242,Z 481.201,A -85,B 0,C 180,E1 -1167.967,E2 -1167.967} C_VEL
LIN {X 0,Y 594.239,Z 482.784,A -85,B 0,C 180,E1 -1169.322,E2 -1169.322} C_VEL
LIN {X 0,Y 594.236,Z 483,A -85,B 0,C 180,E1 -1170,E2 -1170} C_VEL
LIN {X 0,Y 594.247,Z 482.185,A -85,B 0,C 180,E1 -1171.355,E2 -1171.355} C_VEL
LIN {X 0,Y 594.242,Z 481.201,A -85,B 0,C 180,E1 -1172.033,E2 -1172.033} C_VEL
LIN {X 0,Y 594.226,Z 479.81,A -85,B 0,C 180,E1 -1172.712,E2 -1172.712} C_VEL
LIN {X 0,Y 594.289,Z 476.896,A -85,B 0,C 180,E1 -1173.729,E2 -1173.729} C_VEL
LIN {X 0,Y 594.241,Z 472.95,A -85,B 0,C 180,E1 -1174.749,E2 -1174.749} C_VEL
LIN {X 0,Y 594.304,Z 466.878,A -85,B 0,C 180,E1 -1175.939,E2 -1175.939} C_VEL
LIN {X 0,Y 594.309,Z 460.237,A -85,B 0,C 180,E1 -1176.962,E2 -1176.962} C_VEL
LIN {X 0,Y 594.36,Z 451.991,A -85,B 0,C 180,E1 -1177.986,E2 -1177.986} C_VEL
LIN {X 0,Y 594.382,Z 443.539,A -85,B 0,C 180,E1 -1178.842,E2 -1178.842} C_VEL
LIN {X 0,Y 594.432,Z 433.097,A -85,B 0,C 180,E1 -1179.699,E2 -1179.699} C_VEL
LIN {X 0,Y 594.487,Z 422.762,A -85,B 0,C 180,E1 -1180.386,E2 -1180.386} C_VEL
LIN {X 0,Y 594.559,Z 411.741,A -85,B 0,C 180,E1 -1180.972,E2 -1180.972} C_VEL
LIN {X 0,Y 594.575,Z 399.723,A -85,B 0,C 180,E1 -1181.464,E2 -1181.464} C_VEL
LIN {X 0,Y 594.613,Z 386.362,A -85,B 0,C 180,E1 -1181.85,E2 -1181.85} C_VEL
LIN {X 0,Y 594.663,Z 373.105,A -85,B 0,C 180,E1 -1182.087,E2 -1182.087} C_VEL
LIN {X 0,Y 594.617,Z 272.286,A -85,B 0,C 180,E1 -1183.311,E2 -1183.311} C_VEL
LIN {X 0,Y 594.436,Z 270.615,A -85,B 0,C 180,E1 -1183.351,E2 -1183.351} C_VEL
LIN {X 0,Y 594.525,Z 250.066,A -85,B 0,C 180,E1 -1186.128,E2 -1186.128} C_VEL
LIN {X 0,Y 594.631,Z 228.409,A -85,B 0,C 180,E1 -1189.097,E2 -1189.097} C_VEL
LIN {X 0,Y 594.743,Z 209.939,A -85,B 0,C 180,E1 -1191.67,E2 -1191.67} C_VEL
LIN {X 0,Y 594.617,Z 202.04,A -85,B 0,C 180,E1 -1192.791,E2 -1192.791} C_VEL
LIN {X 0,Y 594.336,Z 200.452,A -85,B 0,C 180,E1 -1193.06,E2 -1193.06} C_VEL
LIN {X 0,Y 594.342,Z 200.455,A -85,B 0,C 180,E1 -1195.945,E2 -1195.945} C_VEL
LIN {X 0,Y 594.294,Z 200.455,A -85,B 0,C 180,E1 -1198.231,E2 -1198.231} C_VEL
LIN {X 0,Y 594.352,Z 200.445,A -85,B 0,C 180,E1 -1200.56,E2 -1200.56} C_VEL
LIN {X 0,Y 594.334,Z 200.446,A -85,B 0,C 180,E1 -1202.952,E2 -1202.952} C_VEL
LIN {X 0,Y 594.305,Z 200.454,A -85,B 0,C 180,E1 -1205.411,E2 -1205.411} C_VEL
LIN {X 0,Y 594.31,Z 200.457,A -85,B 0,C 180,E1 -1207.945,E2 -1207.945} C_VEL
LIN {X 0,Y 594.305,Z 200.45,A -85,B 0,C 180,E1 -1210.571,E2 -1210.571} C_VEL
LIN {X 0,Y 594.302,Z 200.45,A -85,B 0,C 180,E1 -1212.844,E2 -1212.844} C_VEL
LIN {X 0,Y 594.329,Z 200.449,A -85,B 0,C 180,E1 -1215.193,E2 -1215.193} C_VEL
LIN {X 0,Y 594.347,Z 200.448,A -85,B 0,C 180,E1 -1218.154,E2 -1218.154} C_VEL
LIN {X 0,Y 594.319,Z 200.45,A -85,B 0,C 180,E1 -1221.188,E2 -1221.188} C_VEL
LIN {X 0,Y 594.335,Z 200.456,A -85,B 0,C 180,E1 -1223.752,E2 -1223.752} C_VEL
LIN {X 0,Y 594.314,Z 200.451,A -85,B 0,C 180,E1 -1226.232,E2 -1226.232} C_VEL
LIN {X 0,Y 594.306,Z 200.449,A -85,B 0,C 180,E1 -1228.644,E2 -1228.644} C_VEL
LIN {X 0,Y 594.335,Z 200.447,A -85,B 0,C 180,E1 -1231.048,E2 -1231.048} C_VEL
LIN {X 0,Y 594.336,Z 200.45,A -85,B 0,C 180,E1 -1234.051,E2 -1234.051} C_VEL
LIN {X 0,Y 594.342,Z 200.446,A -85,B 0,C 180,E1 -1236.291,E2 -1236.291} C_VEL
LIN {X 0,Y 594.363,Z 200.446,A -85,B 0,C 180,E1 -1239.22,E2 -1239.22} C_VEL
LIN {X 0,Y 594.348,Z 200.451,A -85,B 0,C 180,E1 -1241.378,E2 -1241.378} C_VEL
LIN {X 0,Y 594.319,Z 200.449,A -85,B 0,C 180,E1 -1244.215,E2 -1244.215} C_VEL
LIN {X 0,Y 594.328,Z 200.447,A -85,B 0,C 180,E1 -1246.317,E2 -1246.317} C_VEL
LIN {X 0,Y 594.322,Z 200.449,A -85,B 0,C 180,E1 -1248.953,E2 -1248.953} C_VEL
LIN {X 0,Y 594.334,Z 200.452,A -85,B 0,C 180,E1 -1251.839,E2 -1251.839} C_VEL
LIN {X 0,Y 594.325,Z 200.452,A -85,B 0,C 180,E1 -1253.887,E2 -1253.887} C_VEL
LIN {X 0,Y 594.313,Z 200.453,A -85,B 0,C 180,E1 -1255.928,E2 -1255.928} C_VEL
LIN {X 0,Y 594.353,Z 200.447,A -85,B 0,C 180,E1 -1257.963,E2 -1257.963} C_VEL
LIN {X 0,Y 594.37,Z 200.444,A -85,B 0,C 180,E1 -1259.996,E2 -1259.996} C_VEL
LIN {X 0,Y 594.352,Z 200.444,A -85,B 0,C 180,E1 -1262.707,E2 -1262.707} C_VEL
LIN {X 0,Y 594.364,Z 200.452,A -85,B 0,C 180,E1 -1265.424,E2 -1265.424} C_VEL
LIN {X 0,Y 594.325,Z 200.448,A -85,B 0,C 180,E1 -1268.154,E2 -1268.154} C_VEL
LIN {X 0,Y 594.344,Z 200.449,A -85,B 0,C 180,E1 -1271.058,E2 -1271.058} C_VEL
LIN {X 0,Y 594.305,Z 200.45,A -85,B 0,C 180,E1 -1274.147,E2 -1274.147} C_VEL
LIN {X 0,Y 594.312,Z 200.452,A -85,B 0,C 180,E1 -1275.275,E2 -1275.275} C_VEL
LIN {X 0,Y 593.639,Z 200.537,A -85,B 0,C 180,E1 -1275.841,E2 -1275.841} C_VEL
LIN {X 0,Y 590.774,Z 200.892,A -85,B 0,C 180,E1 -1276.759,E2 -1276.759} C_VEL
LIN {X 0,Y 588.362,Z 201.199,A -85,B 0,C 180,E1 -1277.497,E2 -1277.497} C_VEL
LIN {X 0,Y 587.338,Z 201.319,A -85,B 0,C 180,E1 -1278.067,E2 -1278.067} C_VEL
LIN {X 0,Y 587.261,Z 201.327,A -85,B 0,C 180,E1 -1278.26,E2 -1278.26} C_VEL
LIN {X 0,Y 587.3,Z 201.327,A -85,B 0,C 180,E1 -1281.033,E2 -1281.033} C_VEL
LIN {X 0,Y 587.265,Z 201.328,A -85,B 0,C 180,E1 -1284.004,E2 -1284.004} C_VEL
LIN {X 0,Y 587.292,Z 201.323,A -85,B 0,C 180,E1 -1286.275,E2 -1286.275} C_VEL
LIN {X 0,Y 587.307,Z 201.328,A -85,B 0,C 180,E1 -1289.129,E2 -1289.129} C_VEL
LIN {X 0,Y 587.308,Z 201.324,A -85,B 0,C 180,E1 -1291.832,E2 -1291.832} C_VEL
LIN {X 0,Y 587.302,Z 201.322,A -85,B 0,C 180,E1 -1294.343,E2 -1294.343} C_VEL
LIN {X 0,Y 587.299,Z 201.328,A -85,B 0,C 180,E1 -1297.604,E2 -1297.604} C_VEL
LIN {X 0,Y 587.268,Z 201.326,A -85,B 0,C 180,E1 -1300.25,E2 -1300.25} C_VEL
LIN {X 0,Y 587.276,Z 201.333,A -85,B 0,C 180,E1 -1303.116,E2 -1303.116} C_VEL
LIN {X 0,Y 587.269,Z 201.327,A -85,B 0,C 180,E1 -1306.046,E2 -1306.046} C_VEL
LIN {X 0,Y 587.288,Z 201.329,A -85,B 0,C 180,E1 -1308.921,E2 -1308.921} C_VEL
LIN {X 0,Y 587.28,Z 201.33,A -85,B 0,C 180,E1 -1311.518,E2 -1311.518} C_VEL
LIN {X 0,Y 587.306,Z 201.322,A -85,B 0,C 180,E1 -1314.45,E2 -1314.45} C_VEL
LIN {X 0,Y 587.285,Z 201.331,A -85,B 0,C 180,E1 -1317.419,E2 -1317.419} C_VEL
LIN {X 0,Y 587.286,Z 201.325,A -85,B 0,C 180,E1 -1319.828,E2 -1319.828} C_VEL
LIN {X 0,Y 587.288,Z 201.324,A -85,B 0,C 180,E1 -1322.304,E2 -1322.304} C_VEL
LIN {X 0,Y 587.277,Z 201.326,A -85,B 0,C 180,E1 -1324.481,E2 -1324.481} C_VEL
LIN {X 0,Y 587.305,Z 201.327,A -85,B 0,C 180,E1 -1327.485,E2 -1327.485} C_VEL
LIN {X 0,Y 587.285,Z 201.326,A -85,B 0,C 180,E1 -1329.694,E2 -1329.694} C_VEL
LIN {X 0,Y 587.274,Z 201.326,A -85,B 0,C 180,E1 -1331.872,E2 -1331.872} C_VEL
LIN {X 0,Y 587.276,Z 201.325,A -85,B 0,C 180,E1 -1334.024,E2 -1334.024} C_VEL
LIN {X 0,Y 587.305,Z 201.322,A -85,B 0,C 180,E1 -1336.153,E2 -1336.153} C_VEL
LIN {X 0,Y 587.342,Z 201.325,A -85,B 0,C 180,E1 -1338.963,E2 -1338.963} C_VEL
LIN {X 0,Y 587.306,Z 201.323,A -85,B 0,C 180,E1 -1341.744,E2 -1341.744} C_VEL
LIN {X 0,Y 587.268,Z 201.327,A -85,B 0,C 180,E1 -1343.817,E2 -1343.817} C_VEL
LIN {X 0,Y 587.25,Z 201.329,A -85,B 0,C 180,E1 -1345.882,E2 -1345.882} C_VEL
LIN {X 0,Y 587.296,Z 201.323,A -85,B 0,C 180,E1 -1347.943,E2 -1347.943} C_VEL
LIN {X 0,Y 587.345,Z 201.321,A -85,B 0,C 180,E1 -1350.686,E2 -1350.686} C_VEL
LIN {X 0,Y 587.294,Z 201.327,A -85,B 0,C 180,E1 -1353.43,E2 -1353.43} C_VEL
LIN {X 0,Y 587.312,Z 201.324,A -85,B 0,C 180,E1 -1355.493,E2 -1355.493} C_VEL
LIN {X 0,Y 587.321,Z 201.322,A -85,B 0,C 180,E1 -1357.563,E2 -1357.563} C_VEL
LIN {X 0,Y 587.293,Z 201.325,A -85,B 0,C 180,E1 -1360.34,E2 -1360.34} C_VEL
LIN {X 0,Y 587.282,Z 201.328,A -85,B 0,C 180,E1 -1362.439,E2 -1362.439} C_VEL
LIN {X 0,Y 587.317,Z 201.471,A -85,B 0,C 180,E1 -1364.112,E2 -1364.112} C_VEL
LIN {X 0,Y 587.41,Z 212.921,A -85,B 0,C 180,E1 -1366.151,E2 -1366.151} C_VEL
LIN {X 0,Y 587.329,Z 229.497,A -85,B 0,C 180,E1 -1369.057,E2 -1369.057} C_VEL
LIN {X 0,Y 587.312,Z 232.356,A -85,B 0,C 180,E1 -1369.555,E2 -1369.555} C_VEL
LIN {X 0,Y 587.837,Z 238.047,A -85,B 0,C 180,E1 -1369.648,E2 -1369.648} C_VEL
LIN {X 0,Y 587.698,Z 339.416,A -85,B 0,C 180,E1 -1370.909,E2 -1370.909} C_VEL
LIN {X 0,Y 587.651,Z 352.536,A -85,B 0,C 180,E1 -1371.214,E2 -1371.214} C_VEL
LIN {X 0,Y 587.592,Z 365.703,A -85,B 0,C 180,E1 -1371.672,E2 -1371.672} C_VEL
LIN {X 0,Y 587.533,Z 377.389,A -85,B 0,C 180,E1 -1372.227,E2 -1372.227} C_VEL
LIN {X 0,Y 587.453,Z 388.734,A -85,B 0,C 180,E1 -1372.917,E2 -1372.917} C_VEL
LIN {X 0,Y 587.398,Z 399.319,A -85,B 0,C 180,E1 -1373.722,E2 -1373.722} C_VEL
LIN {X 0,Y 587.324,Z 408.55,A -85,B 0,C 180,E1 -1374.591,E2 -1374.591} C_VEL
LIN {X 0,Y 587.267,Z 416.635,A -85,B 0,C 180,E1 -1375.519,E2 -1375.519} C_VEL
LIN {X 0,Y 587.239,Z 423.463,A -85,B 0,C 180,E1 -1376.474,E2 -1376.474} C_VEL
LIN {X 0,Y 587.184,Z 430.335,A -85,B 0,C 180,E1 -1377.677,E2 -1377.677} C_VEL
LIN {X 0,Y 587.155,Z 434.463,A -85,B 0,C 180,E1 -1378.605,E2 -1378.605} C_VEL
LIN {X 0,Y 587.183,Z 438.466,A -85,B 0,C 180,E1 -1379.782,E2 -1379.782} C_VEL
LIN {X 0,Y 587.152,Z 441.182,A -85,B 0,C 180,E1 -1380.976,E2 -1380.976} C_VEL
LIN {X 0,Y 587.135,Z 442.347,A -85,B 0,C 180,E1 -1381.815,E2 -1381.815} C_VEL
LIN {X 0,Y 587.109,Z 442.996,A -85,B 0,C 180,E1 -1383.09,E2 -1383.09} C_VEL
LIN {X 0,Y 587.125,Z 442.286,A -85,B 0,C 180,E1 -1384.328,E2 -1384.328} C_VEL
LIN {X 0,Y 587.136,Z 440.372,A -85,B 0,C 180,E1 -1385.527,E2 -1385.527} C_VEL
LIN {X 0,Y 587.179,Z 437.087,A -85,B 0,C 180,E1 -1386.758,E2 -1386.758} C_VEL
LIN {X 0,Y 587.172,Z 433.045,A -85,B 0,C 180,E1 -1387.828,E2 -1387.828} C_VEL
LIN {X 0,Y 587.187,Z 427.589,A -85,B 0,C 180,E1 -1388.934,E2 -1388.934} C_VEL
LIN {X 0,Y 587.249,Z 420.743,A -85,B 0,C 180,E1 -1390.02,E2 -1390.02} C_VEL
LIN {X 0,Y 587.283,Z 412.415,A -85,B 0,C 180,E1 -1391.079,E2 -1391.079} C_VEL
LIN {X 0,Y 587.373,Z 403.96,A -85,B 0,C 180,E1 -1391.954,E2 -1391.954} C_VEL
LIN {X 0,Y 587.431,Z 394.443,A -85,B 0,C 180,E1 -1392.76,E2 -1392.76} C_VEL
LIN {X 0,Y 587.477,Z 383.604,A -85,B 0,C 180,E1 -1393.505,E2 -1393.505} C_VEL
LIN {X 0,Y 587.564,Z 371.804,A -85,B 0,C 180,E1 -1394.146,E2 -1394.146} C_VEL
LIN {X 0,Y 587.625,Z 359.753,A -85,B 0,C 180,E1 -1394.645,E2 -1394.645} C_VEL
LIN {X 0,Y 587.681,Z 347.217,A -85,B 0,C 180,E1 -1395.017,E2 -1395.017} C_VEL
LIN {X 0,Y 587.741,Z 333.813,A -85,B 0,C 180,E1 -1395.267,E2 -1395.267} C_VEL
LIN {X 0,Y 587.703,Z 234.739,A -85,B 0,C 180,E1 -1396.486,E2 -1396.486} C_VEL
LIN {X 0,Y 587.323,Z 232.324,A -85,B 0,C 180,E1 -1396.541,E2 -1396.541} C_VEL
LIN {X 0,Y 587.433,Z 216.301,A -85,B 0,C 180,E1 -1399.342,E2 -1399.342} C_VEL
LIN {X 0,Y 587.481,Z 203.891,A -85,B 0,C 180,E1 -1401.54,E2 -1401.54} C_VEL
LIN {X 0,Y 587.327,Z 201.323,A -85,B 0,C 180,E1 -1402.048,E2 -1402.048} C_VEL
LIN {X 0,Y 587.325,Z 201.328,A -85,B 0,C 180,E1 -1404.951,E2 -1404.951} C_VEL
LIN {X 0,Y 587.306,Z 201.327,A -85,B 0,C 180,E1 -1407.426,E2 -1407.426} C_VEL
LIN {X 0,Y 587.31,Z 201.322,A -85,B 0,C 180,E1 -1409.835,E2 -1409.835} C_VEL
LIN {X 0,Y 587.317,Z 201.321,A -85,B 0,C 180,E1 -1412.311,E2 -1412.311} C_VEL
LIN {X 0,Y 587.31,Z 201.324,A -85,B 0,C 180,E1 -1414.488,E2 -1414.488} C_VEL
LIN {X 0,Y 587.31,Z 201.324,A -85,B 0,C 180,E1 -1417.491,E2 -1417.491} C_VEL
LIN {X 0,Y 587.3,Z 201.323,A -85,B 0,C 180,E1 -1419.7,E2 -1419.7} C_VEL
LIN {X 0,Y 587.332,Z 201.324,A -85,B 0,C 180,E1 -1422.599,E2 -1422.599} C_VEL
LIN {X 0,Y 587.332,Z 201.319,A -85,B 0,C 180,E1 -1425.747,E2 -1425.747} C_VEL
LIN {X 0,Y 587.372,Z 201.322,A -85,B 0,C 180,E1 -1428.968,E2 -1428.968} C_VEL
LIN {X 0,Y 587.316,Z 201.32,A -85,B 0,C 180,E1 -1431.748,E2 -1431.748} C_VEL
LIN {X 0,Y 587.346,Z 201.322,A -85,B 0,C 180,E1 -1434.511,E2 -1434.511} C_VEL
LIN {X 0,Y 587.343,Z 201.32,A -85,B 0,C 180,E1 -1437.261,E2 -1437.261} C_VEL
LIN {X 0,Y 587.35,Z 201.317,A -85,B 0,C 180,E1 -1440.004,E2 -1440.004} C_VEL
LIN {X 0,Y 587.364,Z 201.324,A -85,B 0,C 180,E1 -1442.747,E2 -1442.747} C_VEL
LIN {X 0,Y 587.32,Z 201.32,A -85,B 0,C 180,E1 -1445.497,E2 -1445.497} C_VEL
LIN {X 0,Y 587.296,Z 201.323,A -85,B 0,C 180,E1 -1447.567,E2 -1447.567} C_VEL
LIN {X 0,Y 587.276,Z 201.325,A -85,B 0,C 180,E1 -1449.648,E2 -1449.648} C_VEL
LIN {X 0,Y 587.31,Z 201.321,A -85,B 0,C 180,E1 -1451.741,E2 -1451.741} C_VEL
LIN {X 0,Y 587.327,Z 201.328,A -85,B 0,C 180,E1 -1454.557,E2 -1454.557} C_VEL
LIN {X 0,Y 587.297,Z 201.323,A -85,B 0,C 180,E1 -1457.411,E2 -1457.411} C_VEL
LIN {X 0,Y 587.295,Z 201.323,A -85,B 0,C 180,E1 -1459.58,E2 -1459.58} C_VEL
LIN {X 0,Y 587.303,Z 201.322,A -85,B 0,C 180,E1 -1461.778,E2 -1461.778} C_VEL
LIN {X 0,Y 587.293,Z 201.329,A -85,B 0,C 180,E1 -1464.764,E2 -1464.764} C_VEL
LIN {X 0,Y 587.298,Z 201.323,A -85,B 0,C 180,E1 -1467.686,E2 -1467.686} C_VEL
LIN {X 0,Y 587.306,Z 201.326,A -85,B 0,C 180,E1 -1470.174,E2 -1470.174} C_VEL
LIN {X 0,Y 587.327,Z 201.32,A -85,B 0,C 180,E1 -1473.112,E2 -1473.112} C_VEL
LIN {X 0,Y 587.271,Z 201.329,A -85,B 0,C 180,E1 -1475.904,E2 -1475.904} C_VEL
LIN {X 0,Y 587.306,Z 201.331,A -85,B 0,C 180,E1 -1478.483,E2 -1478.483} C_VEL
LIN {X 0,Y 587.283,Z 201.325,A -85,B 0,C 180,E1 -1481.164,E2 -1481.164} C_VEL
LIN {X 0,Y 587.302,Z 201.329,A -85,B 0,C 180,E1 -1484.112,E2 -1484.112} C_VEL
LIN {X 0,Y 587.269,Z 201.328,A -85,B 0,C 180,E1 -1486.991,E2 -1486.991} C_VEL
LIN {X 0,Y 587.287,Z 201.329,A -85,B 0,C 180,E1 -1489.987,E2 -1489.987} C_VEL
LIN {X 0,Y 587.308,Z 201.33,A -85,B 0,C 180,E1 -1492.391,E2 -1492.391} C_VEL
LIN {X 0,Y 587.32,Z 201.322,A -85,B 0,C 180,E1 -1495.658,E2 -1495.658} C_VEL
LIN {X 0,Y 587.301,Z 201.334,A -85,B 0,C 180,E1 -1498.23,E2 -1498.23} C_VEL
LIN {X 0,Y 587.297,Z 201.325,A -85,B 0,C 180,E1 -1500.878,E2 -1500.878} C_VEL
LIN {X 0,Y 587.295,Z 201.329,A -85,B 0,C 180,E1 -1503.834,E2 -1503.834} C_VEL
LIN {X 0,Y 587.319,Z 201.412,A -85,B 0,C 180,E1 -1506.822,E2 -1506.822} C_VEL
LIN {X 0,Y 587.823,Z 206.056,A -85,B 0,C 180,E1 -1507.506,E2 -1507.506} C_VEL
LIN {X 0,Y 587.728,Z 225.472,A -85,B 0,C 180,E1 -1510.257,E2 -1510.257} C_VEL
LIN {X 0,Y 587.556,Z 247.478,A -85,B 0,C 180,E1 -1513.318,E2 -1513.318} C_VEL
LIN {X 0,Y 587.43,Z 269.483,A -85,B 0,C 180,E1 -1516.333,E2 -1516.333} C_VEL
LIN {X 0,Y 587.381,Z 270.616,A -85,B 0,C 180,E1 -1516.486,E2 -1516.486} C_VEL
LIN {X 0,Y 587.838,Z 274.752,A -85,B 0,C 180,E1 -1516.563,E2 -1516.563} C_VEL
LIN {X 0,Y 587.72,Z 378.966,A -85,B 0,C 180,E1 -1517.855,E2 -1517.855} C_VEL
LIN {X 0,Y 587.682,Z 392.232,A -85,B 0,C 180,E1 -1518.161,E2 -1518.161} C_VEL
LIN {X 0,Y 587.606,Z 404.635,A -85,B 0,C 180,E1 -1518.585,E2 -1518.585} C_VEL
LIN {X 0,Y 587.53,Z 416.636,A -85,B 0,C 180,E1 -1519.141,E2 -1519.141} C_VEL
LIN {X 0,Y 587.469,Z 428.207,A -85,B 0,C 180,E1 -1519.837,E2 -1519.837} C_VEL
LIN {X 0,Y 587.394,Z 438.602,A -85,B 0,C 180,E1 -1520.618,E2 -1520.618} C_VEL
LIN {X 0,Y 587.31,Z 447.115,A -85,B 0,C 180,E1 -1521.398,E2 -1521.398} C_VEL
LIN {X 0,Y 587.274,Z 454.963,A -85,B 0,C 180,E1 -1522.263,E2 -1522.263} C_VEL
LIN {X 0,Y 587.232,Z 461.471,A -85,B 0,C 180,E1 -1523.127,E2 -1523.127} C_VEL
LIN {X 0,Y 587.236,Z 467.868,A -85,B 0,C 180,E1 -1524.162,E2 -1524.162} C_VEL
LIN {X 0,Y 587.147,Z 472.951,A -85,B 0,C 180,E1 -1525.194,E2 -1525.194} C_VEL
LIN {X 0,Y 587.213,Z 476.896,A -85,B 0,C 180,E1 -1526.226,E2 -1526.226} C_VEL
LIN {X 0,Y 587.132,Z 479.809,A -85,B 0,C 180,E1 -1527.256,E2 -1527.256} C_VEL
LIN {X 0,Y 587.141,Z 481.2,A -85,B 0,C 180,E1 -1527.942,E2 -1527.942} C_VEL
LIN {X 0,Y 587.14,Z 482.785,A -85,B 0,C 180,E1 -1529.314,E2 -1529.314} C_VEL
LIN {X 0,Y 587.137,Z 483,A -85,B 0,C 180,E1 -1530,E2 -1530} C_VEL
LIN {X 0,Y 587.147,Z 482.186,A -85,B 0,C 180,E1 -1531.372,E2 -1531.372} C_VEL
LIN {X 0,Y 587.141,Z 481.201,A -85,B 0,C 180,E1 -1532.058,E2 -1532.058} C_VEL
LIN {X 0,Y 587.132,Z 479.81,A -85,B 0,C 180,E1 -1532.744,E2 -1532.744} C_VEL
LIN {X 0,Y 587.213,Z 476.896,A -85,B 0,C 180,E1 -1533.774,E2 -1533.774} C_VEL
LIN {X 0,Y 587.147,Z 472.95,A -85,B 0,C 180,E1 -1534.806,E2 -1534.806} C_VEL
LIN {X 0,Y 587.217,Z 466.878,A -85,B 0,C 180,E1 -1536.011,E2 -1536.011} C_VEL
LIN {X 0,Y 587.246,Z 460.238,A -85,B 0,C 180,E1 -1537.046,E2 -1537.046} C_VEL
LIN {X 0,Y 587.3,Z 451.992,A -85,B 0,C 180,E1 -1538.083,E2 -1538.083} C_VEL
LIN {X 0,Y 587.344,Z 443.54,A -85,B 0,C 180,E1 -1538.949,E2 -1538.949} C_VEL
LIN {X 0,Y 587.42,Z 433.099,A -85,B 0,C 180,E1 -1539.816,E2 -1539.816} C_VEL
LIN {X 0,Y 587.49,Z 422.761,A -85,B 0,C 180,E1 -1540.511,E2 -1540.511} C_VEL
LIN {X 0,Y 587.57,Z 410.992,A -85,B 0,C 180,E1 -1541.14,E2 -1541.14} C_VEL
LIN {X 0,Y 587.612,Z 398.609,A -85,B 0,C 180,E1 -1541.639,E2 -1541.639} C_VEL
LIN {X 0,Y 587.671,Z 385.446,A -85,B 0,C 180,E1 -1542.014,E2 -1542.014} C_VEL
LIN {X 0,Y 587.742,Z 373.105,A -85,B 0,C 180,E1 -1542.232,E2 -1542.232} C_VEL
LIN {X 0,Y 587.709,Z 272.732,A -85,B 0,C 180,E1 -1543.465,E2 -1543.465} C_VEL
LIN {X 0,Y 587.381,Z 270.615,A -85,B 0,C 180,E1 -1543.514,E2 -1543.514} C_VEL
LIN {X 0,Y 587.546,Z 251.36,A -85,B 0,C 180,E1 -1546.147,E2 -1546.147} C_VEL
LIN {X 0,Y 587.672,Z 229.852,A -85,B 0,C 180,E1 -1549.13,E2 -1549.13} C_VEL
LIN {X 0,Y 587.819,Z 211.233,A -85,B 0,C 180,E1 -1551.754,E2 -1551.754} C_VEL
LIN {X 0,Y 587.617,Z 203.035,A -85,B 0,C 180,E1 -1552.935,E2 -1552.935} C_VEL
LIN {X 0,Y 587.294,Z 201.33,A -85,B 0,C 180,E1 -1553.206,E2 -1553.206} C_VEL
LIN {X 0,Y 587.295,Z 201.329,A -85,B 0,C 180,E1 -1556.166,E2 -1556.166} C_VEL
LIN {X 0,Y 587.297,Z 201.324,A -85,B 0,C 180,E1 -1559.122,E2 -1559.122} C_VEL
LIN {X 0,Y 587.297,Z 201.333,A -85,B 0,C 180,E1 -1561.826,E2 -1561.826} C_VEL
LIN {X 0,Y 587.297,Z 201.325,A -85,B 0,C 180,E1 -1564.339,E2 -1564.339} C_VEL
LIN {X 0,Y 587.266,Z 201.326,A -85,B 0,C 180,E1 -1566.752,E2 -1566.752} C_VEL
LIN {X 0,Y 587.304,Z 201.325,A -85,B 0,C 180,E1 -1569.361,E2 -1569.361} C_VEL
LIN {X 0,Y 587.286,Z 201.329,A -85,B 0,C 180,E1 -1572.1,E2 -1572.1} C_VEL
LIN {X 0,Y 587.277,Z 201.326,A -85,B 0,C 180,E1 -1575.083,E2 -1575.083} C_VEL
LIN {X 0,Y 587.298,Z 201.33,A -85,B 0,C 180,E1 -1577.921,E2 -1577.921} C_VEL
LIN {X 0,Y 587.299,Z 201.322,A -85,B 0,C 180,E1 -1580.635,E2 -1580.635} C_VEL
LIN {X 0,Y 587.262,Z 201.331,A -85,B 0,C 180,E1 -1583.302,E2 -1583.302} C_VEL
LIN {X 0,Y 587.289,Z 201.333,A -85,B 0,C 180,E1 -1585.773,E2 -1585.773} C_VEL
LIN {X 0,Y 587.298,Z 201.325,A -85,B 0,C 180,E1 -1588.226,E2 -1588.226} C_VEL
LIN {X 0,Y 587.294,Z 201.323,A -85,B 0,C 180,E1 -1590.874,E2 -1590.874} C_VEL
LIN {X 0,Y 587.29,Z 201.331,A -85,B 0,C 180,E1 -1593.83,E2 -1593.83} C_VEL
LIN {X 0,Y 587.293,Z 201.323,A -85,B 0,C 180,E1 -1596.737,E2 -1596.737} C_VEL
LIN {X 0,Y 587.296,Z 201.332,A -85,B 0,C 180,E1 -1599.691,E2 -1599.691} C_VEL
LIN {X 0,Y 587.266,Z 201.332,A -85,B 0,C 180,E1 -1601.868,E2 -1601.868} C_VEL
LIN {X 0,Y 587.28,Z 201.328,A -85,B 0,C 180,E1 -1604.021,E2 -1604.021} C_VEL
LIN {X 0,Y 587.314,Z 201.322,A -85,B 0,C 180,E1 -1606.15,E2 -1606.15} C_VEL
LIN {X 0,Y 587.282,Z 201.326,A -85,B 0,C 180,E1 -1608.958,E2 -1608.958} C_VEL
LIN {X 0,Y 587.302,Z 201.329,A -85,B 0,C 180,E1 -1611.74,E2 -1611.74} C_VEL
LIN {X 0,Y 587.284,Z 201.33,A -85,B 0,C 180,E1 -1613.814,E2 -1613.814} C_VEL
LIN {X 0,Y 587.269,Z 201.331,A -85,B 0,C 180,E1 -1615.879,E2 -1615.879} C_VEL
LIN {X 0,Y 587.327,Z 201.323,A -85,B 0,C 180,E1 -1617.939,E2 -1617.939} C_VEL
LIN {X 0,Y 587.341,Z 201.32,A -85,B 0,C 180,E1 -1619.996,E2 -1619.996} C_VEL
LIN {X 0,Y 587.323,Z 201.32,A -85,B 0,C 180,E1 -1622.739,E2 -1622.739} C_VEL
LIN {X 0,Y 587.327,Z 201.33,A -85,B 0,C 180,E1 -1625.489,E2 -1625.489} C_VEL
LIN {X 0,Y 587.292,Z 201.324,A -85,B 0,C 180,E1 -1628.252,E2 -1628.252} C_VEL
LIN {X 0,Y 587.326,Z 201.324,A -85,B 0,C 180,E1 -1631.129,E2 -1631.129} C_VEL
LIN {X 0,Y 587.276,Z 201.326,A -85,B 0,C 180,E1 -1634.231,E2 -1634.231} C_VEL
LIN {X 0,Y 587.296,Z 201.324,A -85,B 0,C 180,E1 -1636.802,E2 -1636.802} C_VEL
LIN {X 0,Y 587.261,Z 201.327,A -85,B 0,C 180,E1 -1638.26,E2 -1638.26} C_VEL
LIN {X 0,Y 586.622,Z 201.409,A -85,B 0,C 180,E1 -1638.832,E2 -1638.832} C_VEL
LIN {X 0,Y 583.816,Z 201.761,A -85,B 0,C 180,E1 -1639.761,E2 -1639.761} C_VEL
LIN {X 0,Y 581.414,Z 202.058,A -85,B 0,C 180,E1 -1640.508,E2 -1640.508} C_VEL
LIN {X 0,Y 580.356,Z 202.193,A -85,B 0,C 180,E1 -1641.085,E2 -1641.085} C_VEL
LIN {X 0,Y 580.255,Z 202.208,A -85,B 0,C 180,E1 -1641.28,E2 -1641.28} C_VEL
LIN {X 0,Y 580.226,Z 202.211,A -85,B 0,C 180,E1 -1643.554,E2 -1643.554} C_VEL
LIN {X 0,Y 580.247,Z 202.201,A -85,B 0,C 180,E1 -1646.328,E2 -1646.328} C_VEL
LIN {X 0,Y 580.257,Z 202.209,A -85,B 0,C 180,E1 -1649.304,E2 -1649.304} C_VEL
LIN {X 0,Y 580.257,Z 202.2,A -85,B 0,C 180,E1 -1652.196,E2 -1652.196} C_VEL
LIN {X 0,Y 580.245,Z 202.202,A -85,B 0,C 180,E1 -1654.692,E2 -1654.692} C_VEL
LIN {X 0,Y 580.253,Z 202.21,A -85,B 0,C 180,E1 -1657.264,E2 -1657.264} C_VEL
LIN {X 0,Y 580.247,Z 202.201,A -85,B 0,C 180,E1 -1660.267,E2 -1660.267} C_VEL
LIN {X 0,Y 580.232,Z 202.204,A -85,B 0,C 180,E1 -1662.702,E2 -1662.702} C_VEL
LIN {X 0,Y 580.217,Z 202.209,A -85,B 0,C 180,E1 -1665.605,E2 -1665.605} C_VEL
LIN {X 0,Y 580.261,Z 202.199,A -85,B 0,C 180,E1 -1668.231,E2 -1668.231} C_VEL
LIN {X 0,Y 580.237,Z 202.208,A -85,B 0,C 180,E1 -1670.963,E2 -1670.963} C_VEL
LIN {X 0,Y 580.243,Z 202.206,A -85,B 0,C 180,E1 -1673.596,E2 -1673.596} C_VEL
LIN {X 0,Y 580.251,Z 202.2,A -85,B 0,C 180,E1 -1676.142,E2 -1676.142} C_VEL
LIN {X 0,Y 580.233,Z 202.204,A -85,B 0,C 180,E1 -1678.613,E2 -1678.613} C_VEL
LIN {X 0,Y 580.245,Z 202.209,A -85,B 0,C 180,E1 -1681.022,E2 -1681.022} C_VEL
LIN {X 0,Y 580.266,Z 202.201,A -85,B 0,C 180,E1 -1683.656,E2 -1683.656} C_VEL
LIN {X 0,Y 580.243,Z 202.202,A -85,B 0,C 180,E1 -1686.441,E2 -1686.441} C_VEL
LIN {X 0,Y 580.235,Z 202.208,A -85,B 0,C 180,E1 -1689.436,E2 -1689.436} C_VEL
LIN {X 0,Y 580.23,Z 202.205,A -85,B 0,C 180,E1 -1691.644,E2 -1691.644} C_VEL
LIN {X 0,Y 580.232,Z 202.204,A -85,B 0,C 180,E1 -1693.825,E2 -1693.825} C_VEL
LIN {X 0,Y 580.226,Z 202.207,A -85,B 0,C 180,E1 -1696.695,E2 -1696.695} C_VEL
LIN {X 0,Y 580.321,Z 202.197,A -85,B 0,C 180,E1 -1698.827,E2 -1698.827} C_VEL
LIN {X 0,Y 580.271,Z 202.2,A -85,B 0,C 180,E1 -1701.643,E2 -1701.643} C_VEL
LIN {X 0,Y 580.23,Z 202.204,A -85,B 0,C 180,E1 -1703.742,E2 -1703.742} C_VEL
LIN {X 0,Y 580.208,Z 202.206,A -85,B 0,C 180,E1 -1705.832,E2 -1705.832} C_VEL
LIN {X 0,Y 580.268,Z 202.198,A -85,B 0,C 180,E1 -1707.918,E2 -1707.918} C_VEL
LIN {X 0,Y 580.314,Z 202.197,A -85,B 0,C 180,E1 -1710.694,E2 -1710.694} C_VEL
LIN {X 0,Y 580.244,Z 202.204,A -85,B 0,C 180,E1 -1713.472,E2 -1713.472} C_VEL
LIN {X 0,Y 580.276,Z 202.199,A -85,B 0,C 180,E1 -1715.56,E2 -1715.56} C_VEL
LIN {X 0,Y 580.276,Z 202.199,A -85,B 0,C 180,E1 -1717.656,E2 -1717.656} C_VEL
LIN {X 0,Y 580.26,Z 202.202,A -85,B 0,C 180,E1 -1720.467,E2 -1720.467} C_VEL
LIN {X 0,Y 580.251,Z 202.206,A -85,B 0,C 180,E1 -1722.592,E2 -1722.592} C_VEL
LIN {X 0,Y 580.282,Z 202.264,A -85,B 0,C 180,E1 -1724.018,E2 -1724.018} C_VEL
LIN {X 0,Y 580.403,Z 211.185,A -85,B 0,C 180,E1 -1725.629,E2 -1725.629} C_VEL
LIN {X 0,Y 580.348,Z 227.511,A -85,B 0,C 180,E1 -1728.535,E2 -1728.535} C_VEL
LIN {X 0,Y 580.26,Z 232.348,A -85,B 0,C 180,E1 -1729.386,E2 -1729.386} C_VEL
LIN {X 0,Y 580.949,Z 237.313,A -85,B 0,C 180,E1 -1729.477,E2 -1729.477} C_VEL
LIN {X 0,Y 580.764,Z 338.957,A -85,B 0,C 180,E1 -1730.752,E2 -1730.752} C_VEL
LIN {X 0,Y 580.712,Z 352.024,A -85,B 0,C 180,E1 -1731.056,E2 -1731.056} C_VEL
LIN {X 0,Y 580.637,Z 364.284,A -85,B 0,C 180,E1 -1731.477,E2 -1731.477} C_VEL
LIN {X 0,Y 580.562,Z 376.39,A -85,B 0,C 180,E1 -1732.04,E2 -1732.04} C_VEL
LIN {X 0,Y 580.443,Z 387.387,A -85,B 0,C 180,E1 -1732.702,E2 -1732.702} C_VEL
LIN {X 0,Y 580.332,Z 398.689,A -85,B 0,C 180,E1 -1733.555,E2 -1733.555} C_VEL
LIN {X 0,Y 580.27,Z 408.885,A -85,B 0,C 180,E1 -1734.523,E2 -1734.523} C_VEL
LIN {X 0,Y 580.205,Z 416.95,A -85,B 0,C 180,E1 -1735.467,E2 -1735.467} C_VEL
LIN {X 0,Y 580.145,Z 422.996,A -85,B 0,C 180,E1 -1736.32,E2 -1736.32} C_VEL
LIN {X 0,Y 580.106,Z 429.301,A -85,B 0,C 180,E1 -1737.41,E2 -1737.41} C_VEL
LIN {X 0,Y 580.066,Z 434.63,A -85,B 0,C 180,E1 -1738.592,E2 -1738.592} C_VEL
LIN {X 0,Y 580.087,Z 438.576,A -85,B 0,C 180,E1 -1739.783,E2 -1739.783} C_VEL
LIN {X 0,Y 580.065,Z 440.659,A -85,B 0,C 180,E1 -1740.671,E2 -1740.671} C_VEL
LIN {X 0,Y 580.031,Z 442.546,A -85,B 0,C 180,E1 -1742.001,E2 -1742.001} C_VEL
LIN {X 0,Y 580.027,Z 442.952,A -85,B 0,C 180,E1 -1743.287,E2 -1743.287} C_VEL
LIN {X 0,Y 580.025,Z 441.856,A -85,B 0,C 180,E1 -1744.713,E2 -1744.713} C_VEL
LIN {X 0,Y 580.04,Z 439.992,A -85,B 0,C 180,E1 -1745.739,E2 -1745.739} C_VEL
LIN {X 0,Y 580.081,Z 436.729,A -85,B 0,C 180,E1 -1746.917,E2 -1746.917} C_VEL
LIN {X 0,Y 580.097,Z 431.821,A -85,B 0,C 180,E1 -1748.16,E2 -1748.16} C_VEL
LIN {X 0,Y 580.151,Z 425.732,A -85,B 0,C 180,E1 -1749.328,E2 -1749.328} C_VEL
LIN {X 0,Y 580.19,Z 419.592,A -85,B 0,C 180,E1 -1750.269,E2 -1750.269} C_VEL
LIN {X 0,Y 580.221,Z 411.047,A -85,B 0,C 180,E1 -1751.334,E2 -1751.334} C_VEL
LIN {X 0,Y 580.354,Z 402.183,A -85,B 0,C 180,E1 -1752.226,E2 -1752.226} C_VEL
LIN {X 0,Y 580.426,Z 392.225,A -85,B 0,C 180,E1 -1753.046,E2 -1753.046} C_VEL
LIN {X 0,Y 580.479,Z 381.581,A -85,B 0,C 180,E1 -1753.757,E2 -1753.757} C_VEL
LIN {X 0,Y 580.594,Z 370.37,A -85,B 0,C 180,E1 -1754.35,E2 -1754.35} C_VEL
LIN {X 0,Y 580.679,Z 358.525,A -85,B 0,C 180,E1 -1754.828,E2 -1754.828} C_VEL
LIN {X 0,Y 580.745,Z 345.447,A -85,B 0,C 180,E1 -1755.205,E2 -1755.205} C_VEL
LIN {X 0,Y 580.836,Z 332.026,A -85,B 0,C 180,E1 -1755.438,E2 -1755.438} C_VEL
LIN {X 0,Y 580.832,Z 235.682,A -85,B 0,C 180,E1 -1756.636,E2 -1756.636} C_VEL
LIN {X 0,Y 580.296,Z 232.411,A -85,B 0,C 180,E1 -1756.692,E2 -1756.692} C_VEL
LIN {X 0,Y 580.425,Z 216.668,A -85,B 0,C 180,E1 -1759.479,E2 -1759.479} C_VEL
LIN {X 0,Y 580.419,Z 203.142,A -85,B 0,C 180,E1 -1761.909,E2 -1761.909} C_VEL
LIN {X 0,Y 580.29,Z 202.2,A -85,B 0,C 180,E1 -1762.11,E2 -1762.11} C_VEL
LIN {X 0,Y 580.277,Z 202.2,A -85,B 0,C 180,E1 -1764.462,E2 -1764.462} C_VEL
LIN {X 0,Y 580.258,Z 202.209,A -85,B 0,C 180,E1 -1766.98,E2 -1766.98} C_VEL
LIN {X 0,Y 580.275,Z 202.202,A -85,B 0,C 180,E1 -1769.43,E2 -1769.43} C_VEL
LIN {X 0,Y 580.285,Z 202.197,A -85,B 0,C 180,E1 -1772.141,E2 -1772.141} C_VEL
LIN {X 0,Y 580.278,Z 202.206,A -85,B 0,C 180,E1 -1774.925,E2 -1774.925} C_VEL
LIN {X 0,Y 580.245,Z 202.201,A -85,B 0,C 180,E1 -1777.952,E2 -1777.952} C_VEL
LIN {X 0,Y 580.29,Z 202.206,A -85,B 0,C 180,E1 -1780.918,E2 -1780.918} C_VEL
LIN {X 0,Y 580.25,Z 202.201,A -85,B 0,C 180,E1 -1783.83,E2 -1783.83} C_VEL
LIN {X 0,Y 580.296,Z 202.195,A -85,B 0,C 180,E1 -1785.987,E2 -1785.987} C_VEL
LIN {X 0,Y 580.33,Z 202.2,A -85,B 0,C 180,E1 -1788.832,E2 -1788.832} C_VEL
LIN {X 0,Y 580.287,Z 202.196,A -85,B 0,C 180,E1 -1791.648,E2 -1791.648} C_VEL
LIN {X 0,Y 580.308,Z 202.198,A -85,B 0,C 180,E1 -1794.444,E2 -1794.444} C_VEL
LIN {X 0,Y 580.312,Z 202.196,A -85,B 0,C 180,E1 -1797.227,E2 -1797.227} C_VEL
LIN {X 0,Y 580.321,Z 202.192,A -85,B 0,C 180,E1 -1800.004,E2 -1800.004} C_VEL
LIN {X 0,Y 580.327,Z 202.201,A -85,B 0,C 180,E1 -1802.78,E2 -1802.78} C_VEL
LIN {X 0,Y 580.287,Z 202.195,A -85,B 0,C 180,E1 -1805.564,E2 -1805.564} C_VEL
LIN {X 0,Y 580.249,Z 202.201,A -85,B 0,C 180,E1 -1807.66,E2 -1807.66} C_VEL
LIN {X 0,Y 580.262,Z 202.205,A -85,B 0,C 180,E1 -1810.471,E2 -1810.471} C_VEL
LIN {X 0,Y 580.285,Z 202.206,A -85,B 0,C 180,E1 -1812.595,E2 -1812.595} C_VEL
LIN {X 0,Y 580.274,Z 202.206,A -85,B 0,C 180,E1 -1814.738,E2 -1814.738} C_VEL
LIN {X 0,Y 580.254,Z 202.2,A -85,B 0,C 180,E1 -1817.629,E2 -1817.629} C_VEL
LIN {X 0,Y 580.273,Z 202.198,A -85,B 0,C 180,E1 -1819.826,E2 -1819.826} C_VEL
LIN {X 0,Y 580.256,Z 202.202,A -85,B 0,C 180,E1 -1822.056,E2 -1822.056} C_VEL
LIN {X 0,Y 580.251,Z 202.208,A -85,B 0,C 180,E1 -1824.718,E2 -1824.718} C_VEL
LIN {X 0,Y 580.241,Z 202.202,A -85,B 0,C 180,E1 -1827.407,E2 -1827.407} C_VEL
LIN {X 0,Y 580.259,Z 202.2,A -85,B 0,C 180,E1 -1829.777,E2 -1829.777} C_VEL
LIN {X 0,Y 580.285,Z 202.202,A -85,B 0,C 180,E1 -1832.204,E2 -1832.204} C_VEL
LIN {X 0,Y 580.269,Z 202.204,A -85,B 0,C 180,E1 -1834.7,E2 -1834.7} C_VEL
LIN {X 0,Y 580.263,Z 202.199,A -85,B 0,C 180,E1 -1837.273,E2 -1837.273} C_VEL
LIN {X 0,Y 580.264,Z 202.202,A -85,B 0,C 180,E1 -1839.937,E2 -1839.937} C_VEL
LIN {X 0,Y 580.252,Z 202.206,A -85,B 0,C 180,E1 -1842.711,E2 -1842.711} C_VEL
LIN {X 0,Y 580.236,Z 202.204,A -85,B 0,C 180,E1 -1845.615,E2 -1845.615} C_VEL
LIN {X 0,Y 580.233,Z 202.212,A -85,B 0,C 180,E1 -1848.228,E2 -1848.228} C_VEL
LIN {X 0,Y 580.239,Z 202.204,A -85,B 0,C 180,E1 -1850.963,E2 -1850.963} C_VEL
LIN {X 0,Y 580.22,Z 202.206,A -85,B 0,C 180,E1 -1853.594,E2 -1853.594} C_VEL
LIN {X 0,Y 580.264,Z 202.208,A -85,B 0,C 180,E1 -1856.143,E2 -1856.143} C_VEL
LIN {X 0,Y 580.243,Z 202.207,A -85,B 0,C 180,E1 -1858.614,E2 -1858.614} C_VEL
LIN {X 0,Y 580.241,Z 202.203,A -85,B 0,C 180,E1 -1861.022,E2 -1861.022} C_VEL
LIN {X 0,Y 580.245,Z 202.205,A -85,B 0,C 180,E1 -1863.677,E2 -1863.677} C_VEL
LIN {X 0,Y 580.266,Z 202.273,A -85,B 0,C 180,E1 -1866.697,E2 -1866.697} C_VEL
LIN {X 0,Y 580.877,Z 207.157,A -85,B 0,C 180,E1 -1867.41,E2 -1867.41} C_VEL
LIN {X 0,Y 580.769,Z 226.767,A -85,B 0,C 180,E1 -1870.195,E2 -1870.195} C_VEL
LIN {X 0,Y 580.564,Z 247.478,A -85,B 0,C 180,E1 -1873.111,E2 -1873.111} C_VEL
LIN {X 0,Y 580.434,Z 269.483,A -85,B 0,C 180,E1 -1876.165,E2 -1876.165} C_VEL
LIN {X 0,Y 580.392,Z 270.616,A -85,B 0,C 180,E1 -1876.32,E2 -1876.32} C_VEL
LIN {X 0,Y 580.939,Z 276.541,A -85,B 0,C 180,E1 -1876.422,E2 -1876.422} C_VEL
LIN {X 0,Y 580.8,Z 378.966,A -85,B 0,C 180,E1 -1877.708,E2 -1877.708} C_VEL
LIN {X 0,Y 580.741,Z 392.232,A -85,B 0,C 180,E1 -1878.017,E2 -1878.017} C_VEL
LIN {X 0,Y 580.641,Z 404.383,A -85,B 0,C 180,E1 -1878.436,E2 -1878.436} C_VEL
LIN {X 0,Y 580.558,Z 416.634,A -85,B 0,C 180,E1 -1879.009,E2 -1879.009} C_VEL
LIN {X 0,Y 580.448,Z 428.206,A -85,B 0,C 180,E1 -1879.713,E2 -1879.713} C_VEL
LIN {X 0,Y 580.345,Z 438.604,A -85,B 0,C 180,E1 -1880.503,E2 -1880.503} C_VEL
LIN {X 0,Y 580.267,Z 447.115,A -85,B 0,C 180,E1 -1881.292,E2 -1881.292} C_VEL
LIN {X 0,Y 580.223,Z 454.963,A -85,B 0,C 180,E1 -1882.168,E2 -1882.168} C_VEL
LIN {X 0,Y 580.155,Z 462.657,A -85,B 0,C 180,E1 -1883.223,E2 -1883.223} C_VEL
LIN {X 0,Y 580.139,Z 469.681,A -85,B 0,C 180,E1 -1884.439,E2 -1884.439} C_VEL
LIN {X 0,Y 580.108,Z 474.373,A -85,B 0,C 180,E1 -1885.484,E2 -1885.484} C_VEL
LIN {X 0,Y 580.123,Z 477.958,A -85,B 0,C 180,E1 -1886.527,E2 -1886.527} C_VEL
LIN {X 0,Y 580.043,Z 479.809,A -85,B 0,C 180,E1 -1887.222,E2 -1887.222} C_VEL
LIN {X 0,Y 580.04,Z 481.199,A -85,B 0,C 180,E1 -1887.917,E2 -1887.917} C_VEL
LIN {X 0,Y 580.04,Z 482.785,A -85,B 0,C 180,E1 -1889.306,E2 -1889.306} C_VEL
LIN {X 0,Y 580.037,Z 483,A -85,B 0,C 180,E1 -1890,E2 -1890} C_VEL
LIN {X 0,Y 580.047,Z 482.186,A -85,B 0,C 180,E1 -1891.389,E2 -1891.389} C_VEL
LIN {X 0,Y 580.04,Z 481.2,A -85,B 0,C 180,E1 -1892.083,E2 -1892.083} C_VEL
LIN {X 0,Y 580.043,Z 479.81,A -85,B 0,C 180,E1 -1892.778,E2 -1892.778} C_VEL
LIN {X 0,Y 580.11,Z 476.896,A -85,B 0,C 180,E1 -1893.821,E2 -1893.821} C_VEL
LIN {X 0,Y 580.053,Z 472.949,A -85,B 0,C 180,E1 -1894.865,E2 -1894.865} C_VEL
LIN {X 0,Y 580.139,Z 466.878,A -85,B 0,C 180,E1 -1896.085,E2 -1896.085} C_VEL
LIN {X 0,Y 580.186,Z 460.239,A -85,B 0,C 180,E1 -1897.132,E2 -1897.132} C_VEL
LIN {X 0,Y 580.251,Z 451.992,A -85,B 0,C 180,E1 -1898.182,E2 -1898.182} C_VEL
LIN {X 0,Y 580.308,Z 443.54,A -85,B 0,C 180,E1 -1899.058,E2 -1899.058} C_VEL
LIN {X 0,Y 580.421,Z 433.101,A -85,B 0,C 180,E1 -1899.936,E2 -1899.936} C_VEL
LIN {X 0,Y 580.493,Z 422.759,A -85,B 0,C 180,E1 -1900.639,E2 -1900.639} C_VEL
LIN {X 0,Y 580.583,Z 411.423,A -85,B 0,C 180,E1 -1901.255,E2 -1901.255} C_VEL
LIN {X 0,Y 580.652,Z 399.775,A -85,B 0,C 180,E1 -1901.741,E2 -1901.741} C_VEL
LIN {X 0,Y 580.738,Z 386.36,A -85,B 0,C 180,E1 -1902.138,E2 -1902.138} C_VEL
LIN {X 0,Y 580.81,Z 373.105,A -85,B 0,C 180,E1 -1902.38,E2 -1902.38} C_VEL
LIN {X 0,Y 580.796,Z 273.405,A -85,B 0,C 180,E1 -1903.62,E2 -1903.62} C_VEL
LIN {X 0,Y 580.392,Z 270.615,A -85,B 0,C 180,E1 -1903.68,E2 -1903.68} C_VEL
LIN {X 0,Y 580.565,Z 248.772,A -85,B 0,C 180,E1 -1906.708,E2 -1906.708} C_VEL
LIN {X 0,Y 580.774,Z 227.923,A -85,B 0,C 180,E1 -1909.641,E2 -1909.641} C_VEL
LIN {X 0,Y 580.89,Z 208.534,A -85,B 0,C 180,E1 -1912.402,E2 -1912.402} C_VEL
LIN {X 0,Y 580.587,Z 203.893,A -85,B 0,C 180,E1 -1913.075,E2 -1913.075} C_VEL
LIN {X 0,Y 580.249,Z 202.209,A -85,B 0,C 180,E1 -1913.34,E2 -1913.34} C_VEL
LIN {X 0,Y 580.245,Z 202.205,A -85,B 0,C 180,E1 -1916.323,E2 -1916.323} C_VEL
LIN {X 0,Y 580.251,Z 202.204,A -85,B 0,C 180,E1 -1919.299,E2 -1919.299} C_VEL
LIN {X 0,Y 580.243,Z 202.208,A -85,B 0,C 180,E1 -1922.019,E2 -1922.019} C_VEL
LIN {X 0,Y 580.256,Z 202.2,A -85,B 0,C 180,E1 -1924.698,E2 -1924.698} C_VEL
LIN {X 0,Y 580.25,Z 202.203,A -85,B 0,C 180,E1 -1927.271,E2 -1927.271} C_VEL
LIN {X 0,Y 580.238,Z 202.205,A -85,B 0,C 180,E1 -1930.262,E2 -1930.262} C_VEL
LIN {X 0,Y 580.21,Z 202.205,A -85,B 0,C 180,E1 -1932.711,E2 -1932.711} C_VEL
LIN {X 0,Y 580.242,Z 202.21,A -85,B 0,C 180,E1 -1935.61,E2 -1935.61} C_VEL
LIN {X 0,Y 580.228,Z 202.206,A -85,B 0,C 180,E1 -1938.224,E2 -1938.224} C_VEL
LIN {X 0,Y 580.233,Z 202.203,A -85,B 0,C 180,E1 -1940.959,E2 -1940.959} C_VEL
LIN {X 0,Y 580.206,Z 202.214,A -85,B 0,C 180,E1 -1943.59,E2 -1943.59} C_VEL
LIN {X 0,Y 580.244,Z 202.204,A -85,B 0,C 180,E1 -1946.138,E2 -1946.138} C_VEL
LIN {X 0,Y 580.232,Z 202.203,A -85,B 0,C 180,E1 -1948.609,E2 -1948.609} C_VEL
LIN {X 0,Y 580.241,Z 202.203,A -85,B 0,C 180,E1 -1951.018,E2 -1951.018} C_VEL
LIN {X 0,Y 580.242,Z 202.212,A -85,B 0,C 180,E1 -1953.673,E2 -1953.673} C_VEL
LIN {X 0,Y 580.247,Z 202.201,A -85,B 0,C 180,E1 -1956.438,E2 -1956.438} C_VEL
LIN {X 0,Y 580.24,Z 202.209,A -85,B 0,C 180,E1 -1959.433,E2 -1959.433} C_VEL
LIN {X 0,Y 580.23,Z 202.213,A -85,B 0,C 180,E1 -1961.641,E2 -1961.641} C_VEL
LIN {X 0,Y 580.235,Z 202.209,A -85,B 0,C 180,E1 -1963.821,E2 -1963.821} C_VEL
LIN {X 0,Y 580.28,Z 202.201,A -85,B 0,C 180,E1 -1965.979,E2 -1965.979} C_VEL
LIN {X 0,Y 580.259,Z 202.2,A -85,B 0,C 180,E1 -1968.823,E2 -1968.823} C_VEL
LIN {X 0,Y 580.276,Z 202.206,A -85,B 0,C 180,E1 -1971.64,E2 -1971.64} C_VEL
LIN {X 0,Y 580.247,Z 202.208,A -85,B 0,C 180,E1 -1973.738,E2 -1973.738} C_VEL
LIN {X 0,Y 580.227,Z 202.209,A -85,B 0,C 180,E1 -1975.829,E2 -1975.829} C_VEL
LIN {X 0,Y 580.3,Z 202.198,A -85,B 0,C 180,E1 -1977.914,E2 -1977.914} C_VEL
LIN {X 0,Y 580.312,Z 202.196,A -85,B 0,C 180,E1 -1979.996,E2 -1979.996} C_VEL
LIN {X 0,Y 580.293,Z 202.196,A -85,B 0,C 180,E1 -1982.773,E2 -1982.773} C_VEL
LIN {X 0,Y 580.29,Z 202.205,A -85,B 0,C 180,E1 -1985.556,E2 -1985.556} C_VEL
LIN {X 0,Y 580.265,Z 202.199,A -85,B 0,C 180,E1 -1988.353,E2 -1988.353} C_VEL
LIN {X 0,Y 580.278,Z 202.203,A -85,B 0,C 180,E1 -1991.187,E2 -1991.187} C_VEL
LIN {X 0,Y 580.242,Z 202.202,A -85,B 0,C 180,E1 -1994.315,E2 -1994.315} C_VEL
LIN {X 0,Y 580.262,Z 202.201,A -85,B 0,C 180,E1 -1996.902,E2 -1996.902} C_VEL
LIN {X 0,Y 580.248,Z 202.204,A -85,B 0,C 180,E1 -1999.819,E2 -1999.819} C_VEL
LIN {X 0,Y 580.255,Z 202.208,A -85,B 0,C 180,E1 -2001.28,E2 -2001.28} C_VEL
LIN {X 0,Y 579.544,Z 202.304,A -85,B 0,C 180,E1 -2001.859,E2 -2001.859} C_VEL
LIN {X 0,Y 576.66,Z 202.661,A -85,B 0,C 180,E1 -2002.799,E2 -2002.799} C_VEL
LIN {X 0,Y 574.257,Z 202.954,A -85,B 0,C 180,E1 -2003.555,E2 -2003.555} C_VEL
LIN {X 0,Y 573.241,Z 203.074,A -85,B 0,C 180,E1 -2004.139,E2 -2004.139} C_VEL
LIN {X 0,Y 573.166,Z 203.083,A -85,B 0,C 180,E1 -2004.337,E2 -2004.337} C_VEL
LIN {X 0,Y 573.182,Z 203.085,A -85,B 0,C 180,E1 -2006.973,E2 -2006.973} C_VEL
LIN {X 0,Y 573.201,Z 203.087,A -85,B 0,C 180,E1 -2009.482,E2 -2009.482} C_VEL
LIN {X 0,Y 573.212,Z 203.078,A -85,B 0,C 180,E1 -2012.641,E2 -2012.641} C_VEL
LIN {X 0,Y 573.164,Z 203.091,A -85,B 0,C 180,E1 -2015.184,E2 -2015.184} C_VEL
LIN {X 0,Y 573.188,Z 203.083,A -85,B 0,C 180,E1 -2017.804,E2 -2017.804} C_VEL
LIN {X 0,Y 573.222,Z 203.076,A -85,B 0,C 180,E1 -2020.524,E2 -2020.524} C_VEL
LIN {X 0,Y 573.203,Z 203.082,A -85,B 0,C 180,E1 -2023.666,E2 -2023.666} C_VEL
LIN {X 0,Y 573.193,Z 203.081,A -85,B 0,C 180,E1 -2026.638,E2 -2026.638} C_VEL
LIN {X 0,Y 573.219,Z 203.083,A -85,B 0,C 180,E1 -2029.474,E2 -2029.474} C_VEL
LIN {X 0,Y 573.181,Z 203.081,A -85,B 0,C 180,E1 -2032.189,E2 -2032.189} C_VEL
LIN {X 0,Y 573.228,Z 203.079,A -85,B 0,C 180,E1 -2034.815,E2 -2034.815} C_VEL
LIN {X 0,Y 573.198,Z 203.081,A -85,B 0,C 180,E1 -2037.767,E2 -2037.767} C_VEL
LIN {X 0,Y 573.213,Z 203.079,A -85,B 0,C 180,E1 -2040.632,E2 -2040.632} C_VEL
LIN {X 0,Y 573.211,Z 203.082,A -85,B 0,C 180,E1 -2043.497,E2 -2043.497} C_VEL
LIN {X 0,Y 573.201,Z 203.079,A -85,B 0,C 180,E1 -2046.134,E2 -2046.134} C_VEL
LIN {X 0,Y 573.205,Z 203.081,A -85,B 0,C 180,E1 -2048.702,E2 -2048.702} C_VEL
LIN {X 0,Y 573.188,Z 203.086,A -85,B 0,C 180,E1 -2051.411,E2 -2051.411} C_VEL
LIN {X 0,Y 573.207,Z 203.08,A -85,B 0,C 180,E1 -2053.621,E2 -2053.621} C_VEL
LIN {X 0,Y 573.184,Z 203.083,A -85,B 0,C 180,E1 -2056.529,E2 -2056.529} C_VEL
LIN {X 0,Y 573.235,Z 203.079,A -85,B 0,C 180,E1 -2059.403,E2 -2059.403} C_VEL
LIN {X 0,Y 573.225,Z 203.076,A -85,B 0,C 180,E1 -2062.249,E2 -2062.249} C_VEL
LIN {X 0,Y 573.239,Z 203.075,A -85,B 0,C 180,E1 -2064.371,E2 -2064.371} C_VEL
LIN {X 0,Y 573.258,Z 203.079,A -85,B 0,C 180,E1 -2067.189,E2 -2067.189} C_VEL
LIN {X 0,Y 573.249,Z 203.073,A -85,B 0,C 180,E1 -2070,E2 -2070} C_VEL
LIN {X 0,Y 573.257,Z 203.078,A -85,B 0,C 180,E1 -2072.811,E2 -2072.811} C_VEL
LIN {X 0,Y 573.241,Z 203.075,A -85,B 0,C 180,E1 -2075.628,E2 -2075.628} C_VEL
LIN {X 0,Y 573.226,Z 203.077,A -85,B 0,C 180,E1 -2077.751,E2 -2077.751} C_VEL
LIN {X 0,Y 573.235,Z 203.079,A -85,B 0,C 180,E1 -2080.597,E2 -2080.597} C_VEL
LIN {X 0,Y 573.203,Z 203.086,A -85,B 0,C 180,E1 -2083.471,E2 -2083.471} C_VEL
LIN {X 0,Y 573.275,Z 203.28,A -85,B 0,C 180,E1 -2083.966,E2 -2083.966} C_VEL
LIN {X 0,Y 573.382,Z 212.474,A -85,B 0,C 180,E1 -2085.643,E2 -2085.643} C_VEL
LIN {X 0,Y 573.293,Z 229.853,A -85,B 0,C 180,E1 -2088.771,E2 -2088.771} C_VEL
LIN {X 0,Y 573.238,Z 232.389,A -85,B 0,C 180,E1 -2089.223,E2 -2089.223} C_VEL
LIN {X 0,Y 574.059,Z 238.38,A -85,B 0,C 180,E1 -2089.325,E2 -2089.325} C_VEL
LIN {X 0,Y 573.822,Z 339.725,A -85,B 0,C 180,E1 -2090.616,E2 -2090.616} C_VEL
LIN {X 0,Y 573.756,Z 353.261,A -85,B 0,C 180,E1 -2090.945,E2 -2090.945} C_VEL
LIN {X 0,Y 573.653,Z 366.188,A -85,B 0,C 180,E1 -2091.413,E2 -2091.413} C_VEL
LIN {X 0,Y 573.55,Z 378.792,A -85,B 0,C 180,E1 -2092.04,E2 -2092.04} C_VEL
LIN {X 0,Y 573.403,Z 390.714,A -85,B 0,C 180,E1 -2092.806,E2 -2092.806} C_VEL
LIN {X 0,Y 573.318,Z 401.342,A -85,B 0,C 180,E1 -2093.674,E2 -2093.674} C_VEL
LIN {X 0,Y 573.216,Z 410.884,A -85,B 0,C 180,E1 -2094.636,E2 -2094.636} C_VEL
LIN {X 0,Y 573.135,Z 418.736,A -85,B 0,C 180,E1 -2095.61,E2 -2095.61} C_VEL
LIN {X 0,Y 573.06,Z 425.809,A -85,B 0,C 180,E1 -2096.698,E2 -2096.698} C_VEL
LIN {X 0,Y 572.996,Z 431.423,A -85,B 0,C 180,E1 -2097.78,E2 -2097.78} C_VEL
LIN {X 0,Y 572.993,Z 436.216,A -85,B 0,C 180,E1 -2098.978,E2 -2098.978} C_VEL
LIN {X 0,Y 572.967,Z 439.71,A -85,B 0,C 180,E1 -2100.191,E2 -2100.191} C_VEL
LIN {X 0,Y 572.945,Z 441.315,A -85,B 0,C 180,E1 -2101.009,E2 -2101.009} C_VEL
LIN {X 0,Y 572.933,Z 442.684,A -85,B 0,C 180,E1 -2102.19,E2 -2102.19} C_VEL
LIN {X 0,Y 572.931,Z 442.903,A -85,B 0,C 180,E1 -2103.503,E2 -2103.503} C_VEL
LIN {X 0,Y 572.94,Z 441.846,A -85,B 0,C 180,E1 -2104.741,E2 -2104.741} C_VEL
LIN {X 0,Y 572.957,Z 439.279,A -85,B 0,C 180,E1 -2106.069,E2 -2106.069} C_VEL
LIN {X 0,Y 572.995,Z 436.108,A -85,B 0,C 180,E1 -2107.143,E2 -2107.143} C_VEL
LIN {X 0,Y 573.02,Z 430.646,A -85,B 0,C 180,E1 -2108.48,E2 -2108.48} C_VEL
LIN {X 0,Y 573.086,Z 424.472,A -85,B 0,C 180,E1 -2109.619,E2 -2109.619} C_VEL
LIN {X 0,Y 573.154,Z 416.593,A -85,B 0,C 180,E1 -2110.763,E2 -2110.763} C_VEL
LIN {X 0,Y 573.206,Z 408.098,A -85,B 0,C 180,E1 -2111.758,E2 -2111.758} C_VEL
LIN {X 0,Y 573.337,Z 398.577,A -85,B 0,C 180,E1 -2112.661,E2 -2112.661} C_VEL
LIN {X 0,Y 573.462,Z 387.306,A -85,B 0,C 180,E1 -2113.521,E2 -2113.521} C_VEL
LIN {X 0,Y 573.601,Z 376.045,A -85,B 0,C 180,E1 -2114.204,E2 -2114.204} C_VEL
LIN {X 0,Y 573.692,Z 363.523,A -85,B 0,C 180,E1 -2114.785,E2 -2114.785} C_VEL
LIN {X 0,Y 573.784,Z 350.552,A -85,B 0,C 180,E1 -2115.225,E2 -2115.225} C_VEL
LIN {X 0,Y 573.867,Z 337.6,A -85,B 0,C 180,E1 -2115.51,E2 -2115.51} C_VEL
LIN {X 0,Y 573.962,Z 236.695,A -85,B 0,C 180,E1 -2116.789,E2 -2116.789} C_VEL
LIN {X 0,Y 573.272,Z 232.386,A -85,B 0,C 180,E1 -2116.867,E2 -2116.867} C_VEL
LIN {X 0,Y 573.388,Z 216.452,A -85,B 0,C 180,E1 -2119.726,E2 -2119.726} C_VEL
LIN {X 0,Y 573.433,Z 204.849,A -85,B 0,C 180,E1 -2121.832,E2 -2121.832} C_VEL
LIN {X 0,Y 573.258,Z 203.076,A -85,B 0,C 180,E1 -2122.154,E2 -2122.154} C_VEL
LIN {X 0,Y 573.241,Z 203.083,A -85,B 0,C 180,E1 -2125.226,E2 -2125.226} C_VEL
LIN {X 0,Y 573.219,Z 203.079,A -85,B 0,C 180,E1 -2127.775,E2 -2127.775} C_VEL
LIN {X 0,Y 573.235,Z 203.079,A -85,B 0,C 180,E1 -2130.639,E2 -2130.639} C_VEL
LIN {X 0,Y 573.241,Z 203.077,A -85,B 0,C 180,E1 -2133.504,E2 -2133.504} C_VEL
LIN {X 0,Y 573.2,Z 203.079,A -85,B 0,C 180,E1 -2136.139,E2 -2136.139} C_VEL
LIN {X 0,Y 573.23,Z 203.082,A -85,B 0,C 180,E1 -2139.178,E2 -2139.178} C_VEL
LIN {X 0,Y 573.206,Z 203.082,A -85,B 0,C 180,E1 -2141.416,E2 -2141.416} C_VEL
LIN {X 0,Y 573.222,Z 203.078,A -85,B 0,C 180,E1 -2143.626,E2 -2143.626} C_VEL
LIN {X 0,Y 573.242,Z 203.074,A -85,B 0,C 180,E1 -2145.811,E2 -2145.811} C_VEL
LIN {X 0,Y 573.264,Z 203.079,A -85,B 0,C 180,E1 -2148.738,E2 -2148.738} C_VEL
LIN {X 0,Y 573.232,Z 203.075,A -85,B 0,C 180,E1 -2151.544,E2 -2151.544} C_VEL
LIN {X 0,Y 573.272,Z 203.073,A -85,B 0,C 180,E1 -2154.376,E2 -2154.376} C_VEL
LIN {X 0,Y 573.28,Z 203.072,A -85,B 0,C 180,E1 -2157.193,E2 -2157.193} C_VEL
LIN {X 0,Y 573.292,Z 203.068,A -85,B 0,C 180,E1 -2160.004,E2 -2160.004} C_VEL
LIN {X 0,Y 573.291,Z 203.077,A -85,B 0,C 180,E1 -2162.815,E2 -2162.815} C_VEL
LIN {X 0,Y 573.256,Z 203.071,A -85,B 0,C 180,E1 -2165.632,E2 -2165.632} C_VEL
LIN {X 0,Y 573.206,Z 203.078,A -85,B 0,C 180,E1 -2167.755,E2 -2167.755} C_VEL
LIN {X 0,Y 573.236,Z 203.083,A -85,B 0,C 180,E1 -2170.601,E2 -2170.601} C_VEL
LIN {X 0,Y 573.207,Z 203.078,A -85,B 0,C 180,E1 -2173.474,E2 -2173.474} C_VEL
LIN {X 0,Y 573.217,Z 203.077,A -85,B 0,C 180,E1 -2175.652,E2 -2175.652} C_VEL
LIN {X 0,Y 573.214,Z 203.077,A -85,B 0,C 180,E1 -2177.853,E2 -2177.853} C_VEL
LIN {X 0,Y 573.231,Z 203.077,A -85,B 0,C 180,E1 -2180.08,E2 -2180.08} C_VEL
LIN {X 0,Y 573.222,Z 203.082,A -85,B 0,C 180,E1 -2182.341,E2 -2182.341} C_VEL
LIN {X 0,Y 573.198,Z 203.079,A -85,B 0,C 180,E1 -2185.416,E2 -2185.416} C_VEL
LIN {X 0,Y 573.22,Z 203.085,A -85,B 0,C 180,E1 -2188.568,E2 -2188.568} C_VEL
LIN {X 0,Y 573.206,Z 203.081,A -85,B 0,C 180,E1 -2190.997,E2 -2190.997} C_VEL
LIN {X 0,Y 573.242,Z 203.073,A -85,B 0,C 180,E1 -2193.523,E2 -2193.523} C_VEL
LIN {X 0,Y 573.183,Z 203.085,A -85,B 0,C 180,E1 -2196.056,E2 -2196.056} C_VEL
LIN {X 0,Y 573.226,Z 203.081,A -85,B 0,C 180,E1 -2198.705,E2 -2198.705} C_VEL
LIN {X 0,Y 573.187,Z 203.082,A -85,B 0,C 180,E1 -2201.59,E2 -2201.59} C_VEL
LIN {X 0,Y 573.214,Z 203.088,A -85,B 0,C 180,E1 -2204.338,E2 -2204.338} C_VEL
LIN {X 0,Y 573.205,Z 203.079,A -85,B 0,C 180,E1 -2207.365,E2 -2207.365} C_VEL
LIN {X 0,Y 573.222,Z 203.082,A -85,B 0,C 180,E1 -2210.573,E2 -2210.573} C_VEL
LIN {X 0,Y 573.203,Z 203.079,A -85,B 0,C 180,E1 -2213.075,E2 -2213.075} C_VEL
LIN {X 0,Y 573.241,Z 203.076,A -85,B 0,C 180,E1 -2215.671,E2 -2215.671} C_VEL
LIN {X 0,Y 573.218,Z 203.088,A -85,B 0,C 180,E1 -2218.184,E2 -2218.184} C_VEL
LIN {X 0,Y 573.22,Z 203.081,A -85,B 0,C 180,E1 -2220.633,E2 -2220.633} C_VEL
LIN {X 0,Y 573.188,Z 203.083,A -85,B 0,C 180,E1 -2223.52,E2 -2223.52} C_VEL
LIN {X 0,Y 573.221,Z 203.085,A -85,B 0,C 180,E1 -2226.56,E2 -2226.56} C_VEL
LIN {X 0,Y 573.928,Z 208.133,A -85,B 0,C 180,E1 -2227.312,E2 -2227.312} C_VEL
LIN {X 0,Y 573.833,Z 228.027,A -85,B 0,C 180,E1 -2230.132,E2 -2230.132} C_VEL
LIN {X 0,Y 573.591,Z 248.302,A -85,B 0,C 180,E1 -2233.016,E2 -2233.016} C_VEL
LIN {X 0,Y 573.404,Z 270.616,A -85,B 0,C 180,E1 -2236.15,E2 -2236.15} C_VEL
LIN {X 0,Y 574.055,Z 276.541,A -85,B 0,C 180,E1 -2236.256,E2 -2236.256} C_VEL
LIN {X 0,Y 573.878,Z 378.965,A -85,B 0,C 180,E1 -2237.558,E2 -2237.558} C_VEL
LIN {X 0,Y 573.801,Z 392.231,A -85,B 0,C 180,E1 -2237.87,E2 -2237.87} C_VEL
LIN {X 0,Y 573.694,Z 404.385,A -85,B 0,C 180,E1 -2238.294,E2 -2238.294} C_VEL
LIN {X 0,Y 573.593,Z 416.644,A -85,B 0,C 180,E1 -2238.874,E2 -2238.874} C_VEL
LIN {X 0,Y 573.438,Z 428.204,A -85,B 0,C 180,E1 -2239.585,E2 -2239.585} C_VEL
LIN {X 0,Y 573.332,Z 438.605,A -85,B 0,C 180,E1 -2240.386,E2 -2240.386} C_VEL
LIN {X 0,Y 573.24,Z 447.116,A -85,B 0,C 180,E1 -2241.185,E2 -2241.185} C_VEL
LIN {X 0,Y 573.162,Z 454.963,A -85,B 0,C 180,E1 -2242.071,E2 -2242.071} C_VEL
LIN {X 0,Y 573.075,Z 462.961,A -85,B 0,C 180,E1 -2243.186,E2 -2243.186} C_VEL
LIN {X 0,Y 573.07,Z 469.681,A -85,B 0,C 180,E1 -2244.37,E2 -2244.37} C_VEL
LIN {X 0,Y 573.029,Z 474.373,A -85,B 0,C 180,E1 -2245.428,E2 -2245.428} C_VEL
